C01365=2140.335600,108.803900,-378.952600,0.257831,3.013758,-90.000210
C01366=2142.949200,108.803900,-378.572900,0.601606,4.635229,-90.000210
C01367=2144.844900,108.803900,-378.971000,-2.778845,5.620716,-90.000210
C01368=2148.346300,108.803900,-378.603900,-0.275020,4.159674,-90.000210
C01369=2149.570000,108.803900,-378.482000,0.870896,2.818952,-90.000210
C01370=2153.470900,108.803900,-378.271600,-1.558445,6.233781,-90.000210
C01371=2155.140500,108.803900,-378.024400,-1.644389,3.477854,-90.000210
C01372=2158.623100,108.803900,-378.023900,-1.644389,8.823550,-90.000210
C01373=2159.706500,108.803900,-378.052300,0.200535,5.133702,-90.000210
C01374=2164.528500,108.803900,-377.988700,-3.924761,4.079460,-90.000210
C01375=2165.061600,108.803900,-377.750400,-1.799087,2.475178,-90.000210
C01376=2169.864400,108.803900,-377.381500,-2.503826,3.529420,-90.000210
C01377=2170.425300,108.803900,-377.373400,-0.068755,3.111161,-90.000210
C01378=2174.112300,108.803900,-377.090200,-0.693279,8.347995,-90.000210
C01379=2174.902100,108.803900,-377.071100,-2.457989,1.495420,-90.000210
C01380=2176.445800,108.803900,-376.837600,-1.151645,6.589015,-90.000210
C01381=2178.587100,108.803900,-377.080000,0.492744,5.546231,-90.000210
C01382=2179.426500,108.803900,-376.837800,-1.403747,4.159674,-90.000210
C01383=2180.476200,108.803900,-376.384800,-1.546986,8.342265,-90.000210
C01384=2181.164700,108.803900,-377.498800,-1.105809,12.839984,-90.000210
C01385=2185.019800,108.803900,-375.142900,-2.314749,16.489725,-90.000210
C01386=2185.530800,108.803900,-375.837200,-0.057296,11.768553,-90.000210
C01387=2188.541900,108.803900,-375.235400,-1.088620,-13.636396,-90.000210
C01388=2185.502100,58.803900,-375.622500,-0.051566,2.028271,-90.000210
C01389=2184.587500,58.803900,-375.704900,-1.157375,9.511099,-90.000210
C01390=2181.334500,58.803900,-375.888300,-0.120321,9.224621,-90.000210
C01391=2180.186000,58.803900,-376.104700,-1.346451,10.616908,-90.000210
C01392=2177.745200,58.803900,-376.686800,1.919409,5.872817,-90.000210
C01393=2175.909400,58.803900,-376.663100,-2.085566,0.280749,-90.000210
C01394=2174.454800,58.803900,-377.270400,-1.896490,10.530964,-90.000210
C01395=2172.787400,58.803900,-376.982500,0.509932,2.314749,-90.000210
C01396=2170.187600,58.803900,-377.417200,3.088243,5.930113,-90.000210
C01397=2168.929400,58.803900,-377.238000,0.807870,1.781899,-90.000210
C01398=2165.565800,58.803900,-377.616500,1.581364,7.792226,-90.000210
C01399=2164.422600,58.803900,-377.925700,0.401070,2.056918,-90.000210
C01400=2160.181900,58.803900,-377.880400,-3.472124,0.567228,-90.000210
C01401=2159.040000,58.803900,-378.155600,1.810547,3.787251,-90.000210
C01402=2155.756900,58.803900,-378.165400,0.618794,5.993139,-90.000210
C01403=2154.515100,58.803900,-378.187200,1.117268,-3.225752,-90.000210
C01404=2150.984900,58.803900,-378.776800,-0.452637,7.333860,-90.000210
C01405=2149.951300,58.803900,-378.829700,2.561121,2.457989,-90.000210
C01406=2145.683000,58.803900,-379.110300,1.793358,0.469825,-90.000210
C01407=2143.964500,58.803900,-379.252700,0.257831,2.045459,-90.000210
C01408=2140.681700,58.803900,-379.571700,-0.401070,3.638282,-90.000210
C01409=2139.364900,58.803900,-379.434900,-2.257454,2.566851,-90.000210
C01410=2135.250600,58.803900,-379.701700,0.166158,5.981679,-90.000210
C01411=2134.565900,58.803900,-379.901400,2.343397,2.274642,-90.000210
C01412=2130.555100,58.803900,-379.773400,0.974028,1.094349,-90.000210
C01413=2128.778000,58.803900,-380.055000,-1.346451,5.099324,-90.000210
C01414=2125.039800,58.803900,-379.997700,-2.005352,1.443854,-90.000210
C01415=2123.450000,58.803900,-380.182100,-2.354857,4.967544,-90.000210
C01416=2120.144500,58.803900,-380.051500,1.065701,4.967544,-90.000210
C01417=2119.439800,58.803900,-380.544400,-3.002299,6.841116,-90.000210
C01418=2115.315400,58.803900,-380.917300,-1.466772,2.755927,-90.000210
C01419=2114.666500,58.803900,-380.805000,-1.220400,4.417505,-90.000210
C01420=2110.782700,58.803900,-381.136300,0.051566,-0.148969,-90.000210
C01421=2109.540100,58.803900,-380.902600,1.226130,4.732631,-90.000210
C01422=2105.405600,58.803900,-381.373500,-0.974028,-0.515662,-90.000210
C01423=2104.154700,58.803900,-381.173700,-0.080214,3.386181,-90.000210
C01424=2100.313800,58.803900,-381.393300,1.443854,-2.939273,-90.000210
C01425=2099.416200,58.803900,-381.361500,3.197104,2.188699,-90.000210
C01426=2095.705700,58.803900,-381.541500,-0.865166,2.297561,-90.000210
C01427=2094.399000,58.803900,-381.243800,-1.902220,10.244485,-90.000210
C01428=2090.482500,58.803900,-381.699500,0.521392,0.538580,-90.000210
C01429=2089.894800,58.803900,-381.726800,-0.343775,7.093218,-90.000210
C01430=2088.622100,58.803900,-381.671700,-4.807116,3.311696,-90.000210
C01431=2085.713800,58.803900,-381.989400,2.509555,1.581364,-90.000210
C01432=2084.932900,58.803900,-382.119500,2.440800,-3.529420,-90.000210
C01433=2083.804500,58.803900,-382.023400,-3.036676,7.293753,-90.000210
C01434=2080.895000,58.803900,-382.327300,-6.864034,7.603150,-90.000210
C01435=2079.430100,58.803900,-382.144100,1.541256,0.137510,-90.000210
C01436=2076.700300,58.803900,-381.799600,-1.140186,-1.695955,-90.000210
C01437=2075.381200,58.803900,-381.594200,2.074107,2.641335,-90.000210
C01438=2074.734300,58.803900,-381.984200,-0.406800,10.204378,-90.000210
C01439=2073.666000,58.803900,-381.686800,1.077161,-1.747521,-90.000210
C01440=2070.998900,58.803900,-382.174100,-2.331938,5.580609,-90.000210
C01441=2069.894200,58.803900,-382.356100,0.022918,2.412152,-90.000210
C01442=2066.142600,58.803900,-381.817600,2.841871,-7.838063,-90.000210
C01443=2065.130800,58.803900,-382.222900,-0.000000,4.973274,-90.000210
C01444=2064.109000,58.803900,-382.313600,0.131780,0.045837,-90.000210
C01445=2059.976500,58.803900,-382.791600,0.017189,2.463719,-90.000210
C01446=2059.344800,58.803900,-382.491600,-1.621471,4.004975,-90.000210
C01447=2055.137600,58.803900,-382.767900,0.246372,0.928192,-90.000210
C01448=2054.262100,58.803900,-382.732000,-1.398017,9.608502,-90.000210
C01449=2050.756100,58.803900,-382.822700,-1.220400,1.799087,-90.000210
C01450=2049.656400,58.803900,-382.466400,-2.268913,4.755550,-90.000210
C01451=2045.238400,58.803900,-383.017300,0.349504,2.372045,-90.000210
C01452=2044.711100,58.803900,-382.562100,3.334614,0.177617,-90.000210
C01453=2040.460400,58.803900,-382.439700,-3.603905,-0.005730,-90.000210
C01454=2039.362700,58.803900,-382.724300,-3.804440,5.242564,-90.000210
C01455=2035.985300,58.803900,-382.893100,0.527121,2.538203,-90.000210
C01456=2034.820500,58.803900,-382.546000,1.346451,3.810169,-90.000210
C01457=2030.644000,58.803900,-382.672600,0.859437,-1.008406,-90.000210
C01458=2030.169900,58.803900,-383.193200,1.621471,1.134456,-90.000210
C01459=2025.187800,58.803900,-382.877900,-0.097403,-1.787628,-90.000210
C01460=2024.574700,58.803900,-383.229400,-0.074485,4.004975,-90.000210
C01461=2020.476400,58.803900,-383.039200,-7.431263,2.692902,-90.000210
C01462=2019.466600,58.803900,-382.959500,2.807493,-3.930490,-90.000210
C01463=2015.631800,58.803900,-382.903800,-2.286102,1.432394,-90.000210
C01464=2015.048100,58.803900,-382.657200,-0.315127,-0.956840,-90.000210
C01465=2010.573400,58.803900,-383.196100,0.435448,-0.481285,-90.000210
C01466=2010.196000,58.803900,-383.078200,1.575634,2.429341,-90.000210
C01467=2005.701400,58.803900,-383.121800,-0.022918,-0.418259,-90.000210
C01468=2004.681200,58.803900,-382.914000,1.650118,-0.464096,-90.000210
C01469=2000.403900,58.803900,-383.270500,2.016811,0.676090,-90.000210
C01470=1999.773000,58.803900,-382.763200,1.363640,-2.314749,-90.000210
C01471=1995.965500,58.803900,-383.525800,1.793358,1.266237,-90.000210
C01472=1994.614700,58.803900,-383.090400,-2.326209,3.873195,-90.000210
C01473=1990.010100,58.803900,-383.727900,2.349127,1.186023,-90.000210
C01474=1989.339500,58.803900,-382.844700,-7.906818,2.383504,-90.000210
C01475=1985.330500,58.803900,-383.000600,-1.541256,4.222699,-90.000210
C01476=1984.855800,58.803900,-383.668700,0.275020,-0.085944,-90.000210
C01477=1980.565200,58.803900,-383.301100,1.713144,0.309397,-90.000210
C01478=1979.406900,58.803900,-383.427700,-3.621093,-0.916732,-90.000210
C01479=1975.633400,58.803900,-383.409200,0.733386,3.426288,-90.000210
C01480=1974.632600,58.803900,-383.625600,-3.472124,-1.008406,-90.000210
C01481=1970.094700,58.803900,-383.404200,-0.297938,3.351803,-90.000210
C01482=1969.228600,58.803900,-383.285200,0.807870,-1.804817,-90.000210
C01483=1965.431900,58.803900,-383.353900,0.985487,0.681820,-90.000210
C01484=1964.322300,58.803900,-383.483100,0.418259,-0.859437,-90.000210
C01485=1960.406200,58.803900,-383.682400,-0.343775,5.815522,-90.000210
C01486=1959.568000,58.803900,-383.464300,0.544310,1.638659,-90.000210
C01487=1955.232300,58.803900,-383.720300,-1.707414,0.166158,-90.000210
C01488=1954.550100,58.803900,-384.072200,0.229183,0.166158,-90.000210
C01489=1950.253700,58.803900,-383.661000,-2.142862,3.959138,-90.000210
C01490=1949.237000,58.803900,-383.741700,-0.991217,-0.796411,-90.000210
C01491=1945.042300,58.803900,-383.696800,0.893814,2.830412,-90.000210
C01492=1944.229400,58.803900,-383.864500,-0.103132,-1.512609,-90.000210
C01493=1940.243800,58.803900,-383.674600,0.853707,0.223454,-90.000210
C01494=1939.598200,58.803900,-383.521800,-2.899166,0.721927,-90.000210
C01495=1934.733400,58.803900,-383.900000,1.180293,0.710468,-90.000210
C01496=1934.150000,58.803900,-383.736200,2.543933,-1.220400,-90.000210
C01497=1929.731700,58.803900,-383.984300,1.650118,-1.088620,-90.000210
C01498=1928.887000,58.803900,-383.919500,1.615741,2.320479,-90.000210
C01499=1925.319200,58.803900,-384.022700,1.294885,0.974028,-90.000210
C01500=1924.421800,58.803900,-383.615600,-0.269290,0.320856,-90.000210
C01501=1920.347700,58.803900,-383.889100,-2.509555,-2.217347,-90.000210
C01502=1918.947700,58.803900,-383.934000,-1.329262,2.979381,-90.000210
C01503=1915.472500,58.803900,-383.526300,2.985110,-2.629876,-90.000210
C01504=1914.276600,58.803900,-383.502500,1.844924,4.486260,-90.000210
C01505=1910.641200,58.803900,-383.604500,-0.395341,-1.466772,-90.000210
C01506=1908.610300,58.803900,-383.777400,0.790682,2.916355,-90.000210
C01507=1904.933000,58.803900,-383.473900,2.326209,0.378152,-90.000210
C01508=1903.988800,58.803900,-383.867400,1.260507,-4.383127,-90.000210
C01509=1899.603400,58.803900,-383.901900,0.211994,-1.203211,-90.000210
C01510=1899.065900,58.803900,-383.767000,-3.466395,-0.664631,-90.000210
C01511=1894.408000,58.803900,-383.572600,-0.996947,0.154699,-90.000210
C01512=1893.986600,58.803900,-383.686900,1.312073,-1.426665,-90.000210
C01513=1890.113800,58.803900,-383.601400,-2.532473,-3.655471,-90.000210
C01514=1885.581400,58.803900,-383.341900,-0.595876,-1.294885,-90.000210
C01515=1885.101800,58.803900,-383.330600,-3.283048,0.360963,-90.000210
C01516=1881.620200,58.803900,-382.819500,1.867842,-2.074107,-90.000210
C01517=1879.575800,58.803900,-383.315200,-2.738738,-4.887330,-90.000210
C01518=1875.961700,58.803900,-383.349800,0.240642,0.063025,-90.000210
C01519=1875.053400,58.803900,-383.258900,-1.105809,1.438124,-90.000210
C01520=1871.217400,58.803900,-383.091600,0.487014,0.847978,-90.000210
C01521=1870.023400,58.803900,-382.821900,-4.852953,-4.520637,-90.000210
C01522=1865.779800,58.803900,-382.711700,-2.028271,-3.305966,-90.000210
C01523=1864.214900,58.803900,-382.880300,0.326586,-1.770440,-90.000210
C01524=1860.166900,58.803900,-382.494200,-1.930868,-0.303668,-90.000210
C01525=1859.143500,58.803900,-382.129700,1.655848,-4.600851,-90.000210
C01526=1856.059600,58.803900,-382.618300,-0.790682,-1.191752,-90.000210
C01527=1854.337100,58.803900,-381.870600,2.005352,1.054242,-90.000210
C01528=1852.620800,58.803900,-382.149500,-0.131780,-5.414451,-90.000210
C01529=1850.548500,58.803900,-382.288500,-0.372423,-3.111161,-90.000210
C01530=1849.250100,58.803900,-382.128200,3.552338,-3.792981,-90.000210
C01531=1847.930100,58.803900,-381.849900,2.263183,-4.480530,-90.000210
C01532=1845.672200,58.803900,-381.812800,-2.223076,-3.838817,-90.000210
C01533=1844.518400,58.803900,-381.759500,-1.054242,-5.786874,-90.000210
C01534=1842.170400,58.803900,-381.737900,0.137510,-1.730333,-90.000210
C01535=1839.610700,58.803900,-381.495500,-0.383882,-3.036676,-90.000210
C01536=1835.873400,58.803900,-381.287400,-0.200535,-4.148214,-90.000210
C01537=1834.250800,58.803900,-381.223900,-0.143239,-4.795657,-90.000210
C01538=1830.424200,58.803900,-381.145200,1.541256,-4.715443,-90.000210
C01539=1829.330400,58.803900,-380.908500,-0.120321,-3.242941,-90.000210
C01540=1825.463600,58.803900,-380.787400,2.727279,-5.345696,-90.000210
C01541=1824.811300,58.803900,-380.790700,0.446907,-3.781521,-90.000210
C01542=1820.697200,58.803900,-380.122400,-4.411775,-2.309020,-90.000210
C01543=1820.073100,58.803900,-380.341800,-1.346451,-3.787251,-90.000210
C01544=1815.208000,58.803900,-379.935100,1.128727,-0.721927,-90.000210
C01545=1813.968500,58.803900,-379.830700,-3.122620,-1.781899,-90.000210
C01546=1810.175300,58.803900,-379.725400,-3.432017,-5.042029,-90.000210
C01547=1809.588700,58.803900,-379.670400,0.847978,-6.038975,-90.000210
C01548=1805.581100,58.803900,-379.087200,-0.458366,-7.156243,-90.000210
C01549=1804.197100,58.803900,-379.105600,4.469071,-6.978626,-90.000210
C01550=1800.624100,58.803900,-378.792900,1.546986,-3.552338,-90.000210
C01551=1800.080000,58.803900,-378.764800,-2.091296,-5.798333,-90.000210
C01552=1795.146200,58.803900,-377.697500,1.472502,-12.330052,-90.000210
C01553=1798.894300,8.803900,-378.601800,-3.489313,-5.557691,-90.000210
C01554=1799.874700,8.803900,-378.703700,-0.905273,-2.790304,-90.000210
C01555=1803.731800,8.803900,-378.851500,-0.527121,-8.542801,-90.000210
C01556=1804.996400,8.803900,-379.130200,1.117268,-9.419426,-90.000210
C01557=1808.212300,8.803900,-379.516200,0.452637,-4.996192,-90.000210
C01558=1810.246100,8.803900,-379.250100,1.002676,-4.365938,-90.000210
C01559=1813.388800,8.803900,-379.809400,-6.302536,0.773493,-90.000210
C01560=1814.666500,8.803900,-379.843100,1.403747,-3.506502,-90.000210
C01561=1817.731100,8.803900,-379.844200,1.518338,-4.308643,-90.000210
C01562=1819.765400,8.803900,-380.143400,1.369369,-0.435448,-90.000210
C01563=1823.736000,8.803900,-380.365700,0.647442,-3.426288,-90.000210
C01564=1825.030000,8.803900,-380.140400,-0.200535,-2.801764,-90.000210
C01565=1829.030600,8.803900,-381.056800,1.294885,-3.724226,-90.000210
C01566=1830.159200,8.803900,-380.847200,0.956840,-3.397640,-90.000210
C01567=1833.665900,8.803900,-381.235100,-1.386558,2.492366,-90.000210
C01568=1834.861100,8.803900,-381.245300,2.841871,-0.750575,-90.000210
C01569=1838.641500,8.803900,-381.487400,1.667307,-4.537826,-90.000210
C01570=1839.725400,8.803900,-381.101400,-1.655848,-0.458366,-90.000210
C01571=1840.896800,8.803900,-381.998000,-2.704361,-9.499640,-90.000210
C01572=1844.249100,8.803900,-381.278200,-1.707414,-1.644389,-90.000210
C01573=1845.828700,8.803900,-381.090700,-0.446907,-2.956462,-90.000210
C01574=1848.645500,8.803900,-381.508500,1.684496,-4.772738,-90.000210
C01575=1849.939500,8.803900,-381.733100,1.758980,2.097026,-90.000210
C01576=1851.853300,8.803900,-381.959200,-0.068755,-1.352180,-90.000210
C01577=1854.092400,8.803900,-382.227200,-0.223454,-2.097026,-90.000210
C01578=1855.033800,8.803900,-381.980700,-1.254778,-1.203211,-90.000210
C01579=1858.951100,8.803900,-381.746000,4.726902,-0.561499,-90.000210
C01580=1860.353300,8.803900,-382.463600,-0.303668,-3.093972,-90.000210
C01581=1861.721700,8.803900,-382.169600,2.022541,0.045837,-90.000210
C01582=1865.128600,8.803900,-382.819200,3.466395,-3.575257,-90.000210
C01583=1866.119700,8.803900,-381.824800,-0.000000,2.435071,-90.000210
C01584=1869.238400,8.803900,-383.038200,0.309397,-4.159674,-90.000210
C01585=1869.781300,8.803900,-382.206600,3.208564,-1.438124,-90.000210
C01586=1874.067800,8.803900,-382.729800,2.137133,2.973651,-90.000210
C01587=1874.982700,8.803900,-382.825800,0.068755,-0.544310,-90.000210
C01588=1877.430700,8.803900,-382.695100,1.415206,-1.976704,-90.000210
C01589=1880.280300,8.803900,-382.513300,-0.876625,-1.690225,-90.000210
C01590=1881.633900,8.803900,-382.741000,-2.629876,-3.575257,-90.000210
C01591=1884.822300,8.803900,-383.129700,-0.338045,-0.962569,-90.000210
C01592=1886.160000,8.803900,-382.472300,-1.546986,2.142862,-90.000210
C01593=1890.121700,8.803900,-383.547500,1.524068,-0.647442,-90.000210
C01594=1891.232400,8.803900,-383.371900,1.002676,-2.320479,-90.000210
C01595=1895.136100,8.803900,-383.093500,-2.074107,0.790682,-90.000210
C01596=1896.427800,8.803900,-383.638300,3.970598,-3.477854,-90.000210
C01597=1899.180000,8.803900,-383.160600,0.068755,-1.254778,-90.000210
C01598=1900.888600,8.803900,-382.681400,3.134079,-2.870519,-90.000210
C01599=1904.903400,8.803900,-383.065000,1.249048,0.475555,-90.000210
C01600=1905.816200,8.803900,-382.772800,2.956462,-0.011459,-90.000210
C01601=1909.631700,8.803900,-382.819700,-2.647065,2.612688,-90.000210
C01602=1914.174000,8.803900,-382.556800,5.878547,0.372423,-90.000210
C01603=1915.668900,8.803900,-383.397100,4.348750,-1.575634,-90.000210
C01604=1918.191500,8.803900,-382.853800,-0.956840,0.412530,-90.000210
C01605=1920.545000,8.803900,-383.109600,1.581364,0.189076,-90.000210
C01606=1923.828600,8.803900,-383.561000,-0.326586,2.011082,-90.000210
C01607=1925.621600,8.803900,-383.491300,2.818952,0.693279,-90.000210
C01608=1928.924300,8.803900,-383.132100,4.153944,2.480907,-90.000210
C01609=1930.221500,8.803900,-383.050700,3.586716,-0.676090,-90.000210
C01610=1934.139500,8.803900,-382.735300,1.976704,0.991217,-90.000210
C01611=1935.506700,8.803900,-382.861000,4.451882,-4.927437,-90.000210
C01612=1938.911000,8.803900,-382.668700,5.712389,3.242941,-90.000210
C01613=1939.988300,8.803900,-382.986500,2.079837,-6.858305,-90.000210
C01614=1944.067300,8.803900,-382.539000,0.515662,-1.019865,-90.000210
C01615=1945.073200,8.803900,-381.750700,3.472124,-2.394964,-90.000210
C01616=1948.562000,8.803900,-383.489800,5.826981,-3.884654,-90.000210
C01617=1949.549500,8.803900,-383.018800,-0.739116,1.799087,-90.000210
C01618=1951.671600,8.803900,-381.909100,2.876248,0.607335,-90.000210
C01619=1954.708200,8.803900,-382.811500,-0.464096,1.008406,-90.000210
C01620=1956.281200,8.803900,-382.140300,1.506879,-0.017189,-90.000210
C01621=1959.804800,8.803900,-382.649900,-0.143239,3.552338,-90.000210
C01622=1960.634200,8.803900,-382.671200,3.919031,3.019488,-90.000210
C01623=1964.757100,8.803900,-383.227900,1.552716,0.859437,-90.000210
C01624=1965.783600,8.803900,-382.461700,-0.206265,1.564175,-90.000210
C01625=1969.332500,8.803900,-382.489900,-2.515285,-1.753251,-90.000210
C01626=1970.399000,8.803900,-382.187200,4.486260,1.495420,-90.000210
C01627=1974.685600,8.803900,-382.745700,2.154321,3.036676,-90.000210
C01628=1975.213800,8.803900,-382.463300,2.755927,-0.051566,-90.000210
C01629=1979.096500,8.803900,-383.224900,-0.572958,6.216592,-90.000210
C01630=1980.965400,8.803900,-382.278900,5.219646,-0.813600,-90.000210
C01631=1983.944900,8.803900,-382.980900,-3.460665,2.904896,-90.000210
C01632=1985.069100,8.803900,-383.157900,2.194428,-5.305589,-90.000210
C01633=1988.765800,8.803900,-382.456300,-0.234913,-2.028271,-90.000210
C01634=1989.888800,8.803900,-382.090400,1.856383,1.432394,-90.000210
C01635=1990.341500,8.803900,-382.930800,1.409476,4.996192,-90.000210
C01636=1993.928900,8.803900,-382.864700,-0.756304,-2.830412,-90.000210
C01637=1995.346700,8.803900,-383.412200,2.807493,4.268536,-90.000210
C01638=1999.376500,8.803900,-382.764300,4.635229,4.555014,-90.000210
C01639=1999.957200,8.803900,-382.491700,1.478231,1.352180,-90.000210
C01640=2001.129100,8.803900,-381.640100,-6.130648,0.487014,-90.000210
C01641=2003.744400,8.803900,-383.015300,-6.291077,4.056541,-90.000210
C01642=2005.057700,8.803900,-382.069000,-0.687549,6.881223,-90.000210
C01643=2008.712000,8.803900,-382.085600,4.812845,1.403747,-90.000210
C01644=2009.806200,8.803900,-382.878700,-0.481285,5.076406,-90.000210
C01645=2012.925600,8.803900,-381.918700,-1.856383,-0.968299,-90.000210
C01646=2015.064200,8.803900,-382.624000,1.438124,-0.189076,-90.000210
C01647=2016.149900,8.803900,-382.482500,-4.320102,4.440423,-90.000210
C01648=2018.113800,8.803900,-382.473600,4.566474,2.973651,-90.000210
C01649=2019.538000,8.803900,-382.127700,1.340721,2.309020,-90.000210
C01650=2020.615000,8.803900,-382.598900,-0.103132,-2.853330,-90.000210
C01651=2023.397600,8.803900,-381.921300,2.268913,6.864034,-90.000210
C01652=2025.430500,8.803900,-381.853800,-0.452637,8.823550,-90.000210
C01653=2026.143200,8.803900,-382.299400,-1.094349,-6.170755,-90.000210
C01654=2029.744600,8.803900,-381.628100,3.506502,-0.080214,-90.000210
C01655=2030.943400,8.803900,-382.368600,1.329262,-2.320479,-90.000210
C01656=2033.843600,8.803900,-381.831700,-4.915978,1.059972,-90.000210
C01657=2035.120700,8.803900,-381.854300,3.191375,1.632930,-90.000210
C01658=2036.216200,8.803900,-381.666200,2.664254,1.254778,-90.000210
C01659=2039.656600,8.803900,-382.222300,2.114214,1.037054,-90.000210
C01660=2040.336700,8.803900,-382.027300,4.623769,3.930490,-90.000210
C01661=2044.682000,8.803900,-381.296300,0.974028,0.750575,-90.000210
C01662=2045.132200,8.803900,-382.311400,1.157375,2.549662,-90.000210
C01663=2046.168000,8.803900,-382.433100,-0.922462,0.716197,-90.000210
C01664=2049.178300,8.803900,-382.426800,0.905273,7.431263,-90.000210
C01665=2050.186200,8.803900,-381.789600,1.650118,3.878924,-90.000210
C01666=2051.798900,8.803900,-381.716500,0.481285,5.958761,-90.000210
C01667=2053.688400,8.803900,-382.030900,1.724603,2.137133,-90.000210
C01668=2054.878700,8.803900,-381.594000,1.363640,2.784575,-90.000210
C01669=2056.375300,8.803900,-381.770500,0.951110,0.137510,-90.000210
C01670=2058.327500,8.803900,-381.651900,2.675713,-5.867088,-90.000210
C01671=2059.785600,8.803900,-382.200000,0.154699,-0.269290,-90.000210
C01672=2061.250400,8.803900,-381.756800,3.214293,2.114214,-90.000210
C01673=2063.874300,8.803900,-382.207100,-3.644012,1.569904,-90.000210
C01674=2065.184100,8.803900,-382.199200,0.721927,-0.825059,-90.000210
C01675=2066.546900,8.803900,-382.027600,1.564175,-0.080214,-90.000210
C01676=2069.277800,8.803900,-381.350500,-1.226130,-1.449583,-90.000210
C01677=2070.702300,8.803900,-381.843300,0.979758,4.102378,-90.000210
C01678=2071.873400,8.803900,-381.587100,-0.028648,7.522936,-90.000210
C01679=2074.360300,8.803900,-381.986800,1.334992,2.561121,-90.000210
C01680=2075.422300,8.803900,-381.676700,2.011082,7.786496,-90.000210
C01681=2078.932700,8.803900,-381.534300,3.145538,-1.002676,-90.000210
C01682=2079.949400,8.803900,-381.507400,2.635606,-5.305589,-90.000210
C01683=2084.420700,8.803900,-381.675300,4.354479,-3.844547,-90.000210
C01684=2085.146700,8.803900,-381.581600,1.913679,2.985110,-90.000210
C01685=2087.746400,8.803900,-381.366900,0.498473,-0.229183,-90.000210
C01686=2089.249100,8.803900,-380.882100,1.770440,2.859059,-90.000210
C01687=2090.194300,8.803900,-382.156400,2.773116,2.372045,-90.000210
C01688=2094.465100,8.803900,-380.936300,-2.423611,2.945003,-90.000210
C01689=2096.081700,8.803900,-381.151500,2.257454,-1.380828,-90.000210
C01690=2099.895500,8.803900,-381.059100,1.042783,-0.951110,-90.000210
C01691=2101.198000,8.803900,-380.864700,2.372045,9.516829,-90.000210
C01692=2105.068100,8.803900,-381.276200,4.062271,4.360209,-90.000210
C01693=2106.438600,8.803900,-380.837900,-0.613065,1.655848,-90.000210
C01694=2109.528900,8.803900,-380.861000,0.704738,1.449583,-90.000210
C01695=2110.846600,8.803900,-380.588700,0.108862,7.041651,-90.000210
C01696=2114.640100,8.803900,-380.177100,-0.217724,2.503826,-90.000210
C01697=2115.458000,8.803900,-380.384400,-0.017189,6.205133,-90.000210
C01698=2119.588600,8.803900,-379.801400,1.088620,1.220400,-90.000210
C01699=2121.498600,8.803900,-379.873500,2.847600,2.354857,-90.000210
C01700=2124.614600,8.803900,-379.701300,-0.297938,0.103132,-90.000210
C01701=2126.311200,8.803900,-379.634300,1.363640,6.686417,-90.000210
C01702=2130.106600,8.803900,-379.760800,0.802141,2.309020,-90.000210
C01703=2133.256100,8.803900,-379.607200,-1.140186,3.082513,-90.000210
C01704=2135.454200,8.803900,-379.716100,1.466772,5.603527,-90.000210
C01705=2138.900600,8.803900,-379.399900,-0.974028,1.856383,-90.000210
C01706=2140.496400,8.803900,-379.454700,1.827735,1.902220,-90.000210
C01707=2143.219500,8.803900,-379.253800,-1.134456,5.614986,-90.000210
C01708=2144.888700,8.803900,-378.834900,-3.197104,6.652040,-90.000210
C01709=2148.266900,8.803900,-379.009800,2.274642,2.102755,-90.000210
C01710=2149.837900,8.803900,-378.563700,0.704738,0.779223,-90.000210
C01711=2154.077000,8.803900,-378.213200,1.558445,4.589392,-90.000210
C01712=2155.082100,8.803900,-378.577300,-0.063025,6.543178,-90.000210
C01713=2158.906100,8.803900,-377.860000,-1.873572,3.374721,-90.000210
C01714=2160.225200,8.803900,-378.014100,-1.948057,3.093972,-90.000210
C01715=2163.890600,8.803900,-377.623900,0.647442,5.614986,-90.000210
C01716=2164.880600,8.803900,-377.783800,1.621471,3.844547,-90.000210
C01717=2169.386500,8.803900,-377.358800,-4.262806,2.074107,-90.000210
C01718=2170.175100,8.803900,-377.246600,-1.489690,0.383882,-90.000210
C01719=2171.774900,8.803900,-376.772400,-2.796034,6.193674,-90.000210
C01720=2174.349300,8.803900,-377.086400,0.017189,4.658147,-90.000210
C01721=2175.360200,8.803900,-377.013800,1.913679,6.674958,-90.000210
C01722=2177.008300,8.803900,-377.163000,-7.454181,1.896490,-90.000210
C01723=2180.561900,8.803900,-376.316900,-0.171887,10.043950,-90.000210
C01724=2181.078100,8.803900,-376.110500,-2.286102,5.076406,-90.000210
C01725=2184.526000,8.803900,-375.725500,-4.314372,8.307888,-90.000210
C01726=2185.880000,-41.196100,-375.195400,-1.117268,8.600097,-90.000210
C01727=2184.495800,-41.196100,-375.702000,-1.524068,7.448451,-90.000210
C01728=2181.254800,-41.196100,-376.002700,-1.180293,5.133702,-90.000210
C01729=2179.901600,-41.196100,-376.252500,-4.881600,5.953031,-90.000210
C01730=2177.291700,-41.196100,-376.736900,-0.504203,5.431640,-90.000210
C01731=2174.987800,-41.196100,-377.102500,-0.263561,6.405668,-90.000210
C01732=2173.467500,-41.196100,-377.244300,-0.017189,6.365561,-90.000210
C01733=2170.873200,-41.196100,-376.921900,-0.349504,3.712767,-90.000210
C01734=2169.363500,-41.196100,-377.460900,-0.211994,7.127595,-90.000210
C01735=2166.065700,-41.196100,-377.214200,1.438124,5.500395,-90.000210
C01736=2165.275200,-41.196100,-377.323000,0.108862,3.432017,-90.000210
C01737=2163.485000,-41.196100,-377.080300,0.819330,6.331184,-90.000210
C01738=2160.102500,-41.196100,-377.738500,1.197482,2.916355,-90.000210
C01739=2158.853300,-41.196100,-377.593900,-1.128727,2.068378,-90.000210
C01740=2155.073000,-41.196100,-378.064900,1.369369,1.925138,-90.000210
C01741=2153.724200,-41.196100,-377.850000,1.352180,2.028271,-90.000210
C01742=2150.349000,-41.196100,-378.400400,0.762034,2.979381,-90.000210
C01743=2149.136700,-41.196100,-377.910500,3.116890,3.678389,-90.000210
C01744=2145.160300,-41.196100,-378.700300,1.655848,3.168457,-90.000210
C01745=2144.326800,-41.196100,-378.466200,1.690225,3.919031,-90.000210
C01746=2140.135800,-41.196100,-378.318400,-1.025594,1.145916,-90.000210
C01747=2138.981500,-41.196100,-379.103600,0.011459,2.068378,-90.000210
C01748=2135.291100,-41.196100,-378.850600,3.271589,3.071054,-90.000210
C01749=2133.841500,-41.196100,-379.406100,0.171887,0.177617,-90.000210
C01750=2130.488700,-41.196100,-378.890300,4.148214,2.584040,-90.000210
C01751=2128.923200,-41.196100,-379.018600,1.799087,7.356778,-90.000210
C01752=2125.737900,-41.196100,-379.393600,3.489313,0.452637,-90.000210
C01753=2123.975700,-41.196100,-378.591300,2.595499,1.839195,-90.000210
C01754=2120.075600,-41.196100,-379.170500,-0.607335,2.309020,-90.000210
C01755=2118.901600,-41.196100,-379.712800,0.916732,4.818575,-90.000210
C01756=2114.735000,-41.196100,-380.002700,-3.317426,-0.126051,-90.000210
C01757=2113.577900,-41.196100,-379.959100,2.962192,-3.260130,-90.000210
C01758=2110.098400,-41.196100,-379.433600,10.227297,3.867465,-90.000210
C01759=2109.561500,-41.196100,-379.487300,3.197104,-2.429341,-90.000210
C01760=2105.376800,-41.196100,-380.509000,4.744091,3.500772,-90.000210
C01761=2104.898100,-41.196100,-379.374400,1.443854,2.967921,-90.000210
C01762=2100.737400,-41.196100,-379.764200,1.352180,-0.045837,-90.000210
C01763=2099.790300,-41.196100,-380.834500,-1.472502,0.229183,-90.000210
C01764=2095.224100,-41.196100,-380.131200,4.612310,2.750197,-90.000210
C01765=2093.930100,-41.196100,-380.331700,1.604282,7.585961,-90.000210
C01766=2089.893200,-41.196100,-380.417300,3.397640,4.761279,-90.000210
C01767=2089.258900,-41.196100,-380.773800,0.779223,-1.925138,-90.000210
C01768=2085.330100,-41.196100,-380.757400,0.790682,0.819330,-90.000210
C01769=2083.879100,-41.196100,-379.511000,3.019488,-1.398017,-90.000210
C01770=2079.836600,-41.196100,-380.416000,0.624524,0.315127,-90.000210
C01771=2079.038700,-41.196100,-380.368400,2.056918,-1.879302,-90.000210
C01772=2074.672000,-41.196100,-379.861700,3.798710,2.498096,-90.000210
C01773=2074.092400,-41.196100,-380.658000,7.047381,8.244863,-90.000210
C01774=2070.056600,-41.196100,-379.715000,-0.464096,3.156997,-90.000210
C01775=2069.076500,-41.196100,-380.400900,-0.326586,-1.277696,-90.000210
C01776=2065.277900,-41.196100,-380.250600,-0.567228,3.277319,-90.000210
C01777=2063.880600,-41.196100,-379.731600,2.251724,-1.380828,-90.000210
C01778=2060.201500,-41.196100,-379.972500,1.163104,-1.231859,-90.000210
C01779=2059.099600,-41.196100,-380.740700,8.227674,1.380828,-90.000210
C01780=2055.123100,-41.196100,-380.849500,3.288778,0.349504,-90.000210
C01781=2053.996000,-41.196100,-380.050500,6.755172,-2.223076,-90.000210
C01782=2049.819700,-41.196100,-380.443700,5.935843,-0.068755,-90.000210
C01783=2049.134800,-41.196100,-381.700300,0.022918,5.660823,-90.000210
C01784=2045.224000,-41.196100,-381.245000,5.523313,1.959516,-90.000210
C01785=2044.771200,-41.196100,-380.905500,-4.027893,-0.074485,-90.000210
C01786=2040.257500,-41.196100,-381.458500,1.094349,4.463341,-90.000210
C01787=2039.336100,-41.196100,-379.745600,0.888085,1.753251,-90.000210
C01788=2035.560200,-41.196100,-380.149800,0.727656,-3.237212,-90.000210
C01789=2033.515600,-41.196100,-381.337000,1.014135,-2.773116,-90.000210
C01790=2029.970400,-41.196100,-381.111700,4.875871,2.091296,-90.000210
C01791=2028.017600,-41.196100,-380.702300,0.750575,-0.905273,-90.000210
C01792=2025.281000,-41.196100,-380.401200,5.380074,-0.429718,-90.000210
C01793=2023.851300,-41.196100,-380.213200,0.481285,-2.435071,-90.000210
C01794=2019.728100,-41.196100,-380.300400,2.412152,-2.400693,-90.000210
C01795=2019.058600,-41.196100,-381.536000,1.764710,2.595499,-90.000210
C01796=2014.946900,-41.196100,-380.978700,1.186023,-0.487014,-90.000210
C01797=2010.390000,-41.196100,-380.567500,-1.638659,5.334237,-90.000210
C01798=2009.731700,-41.196100,-381.456000,3.964868,1.506879,-90.000210
C01799=2006.217700,-41.196100,-381.020200,0.154699,3.993516,-90.000210
C01800=2004.385900,-41.196100,-380.094900,1.220400,2.790304,-90.000210
C01801=2001.248400,-41.196100,-381.863700,6.669229,5.082136,-90.000210
C01802=2000.379500,-41.196100,-380.943500,5.586339,0.550039,-90.000210
C01803=1997.761400,-41.196100,-382.132400,2.211617,-0.171887,-90.000210
C01804=1995.113800,-41.196100,-381.971700,0.257831,3.105431,-90.000210
C01805=1994.652900,-41.196100,-379.974000,2.188699,1.707414,-90.000210
C01806=1989.787700,-41.196100,-381.076400,2.217347,-1.122997,-90.000210
C01807=1989.016100,-41.196100,-379.930100,2.349127,0.389611,-90.000210
C01808=1986.291800,-41.196100,-381.148200,-1.168834,-0.704738,-90.000210
C01809=1984.627600,-41.196100,-380.667900,5.746767,2.343397,-90.000210
C01810=1980.711100,-41.196100,-381.395000,3.093972,-0.481285,-90.000210
C01811=1980.047300,-41.196100,-381.569600,2.016811,-4.279995,-90.000210
C01812=1976.640500,-41.196100,-382.374000,6.972896,-1.340721,-90.000210
C01813=1975.100000,-41.196100,-380.121300,-2.784575,0.137510,-90.000210
C01814=1973.698600,-41.196100,-381.294000,-0.080214,5.609257,-90.000210
C01815=1970.010500,-41.196100,-380.203500,9.316294,-2.515285,-90.000210
C01816=1968.613500,-41.196100,-382.095800,-1.031324,1.844924,-90.000210
C01817=1966.022300,-41.196100,-381.592700,3.999245,2.543933,-90.000210
C01818=1964.655500,-41.196100,-380.029600,2.131403,1.839195,-90.000210
C01819=1960.547600,-41.196100,-380.255200,2.165780,1.718873,-90.000210
C01820=1959.422400,-41.196100,-380.031900,8.519882,-1.867842,-90.000210
C01821=1957.473800,-41.196100,-382.205800,3.099702,-0.779223,-90.000210
C01822=1955.043700,-41.196100,-381.735600,4.394586,0.137510,-90.000210
C01823=1954.062100,-41.196100,-381.684000,6.554637,1.541256,-90.000210
C01824=1950.141700,-41.196100,-380.586400,4.795657,0.825059,-90.000210
C01825=1949.476100,-41.196100,-381.977900,1.816276,-8.233404,-90.000210
C01826=1945.507800,-41.196100,-381.667900,1.277696,5.792603,-90.000210
C01827=1944.984400,-41.196100,-381.700800,3.386181,2.412152,-90.000210
C01828=1943.695100,-41.196100,-382.237100,-0.011459,2.377775,-90.000210
C01829=1941.079500,-41.196100,-381.081000,1.804817,4.463341,-90.000210
C01830=1939.451900,-41.196100,-380.357700,0.538580,3.781521,-90.000210
C01831=1935.406000,-41.196100,-381.487800,2.228806,-1.690225,-90.000210
C01832=1934.176300,-41.196100,-380.632300,5.746767,-0.762034,-90.000210
C01833=1930.488600,-41.196100,-381.185900,6.159296,-2.417882,-90.000210
C01834=1929.880500,-41.196100,-381.659800,-1.684496,0.492744,-90.000210
C01835=1926.074600,-41.196100,-380.394200,0.842248,4.211240,-90.000210
C01836=1924.491200,-41.196100,-380.870900,6.972896,-0.097403,-90.000210
C01837=1920.888500,-41.196100,-380.599800,4.320102,4.148214,-90.000210
C01838=1920.372900,-41.196100,-381.287800,7.058840,-6.858305,-90.000210
C01839=1919.171800,-41.196100,-382.295300,0.005730,2.446530,-90.000210
C01840=1915.534400,-41.196100,-381.857100,-6.995815,13.229595,-90.000210
C01841=1914.581800,-41.196100,-381.964100,10.513776,-7.540125,-90.000210
C01842=1910.831800,-41.196100,-382.252200,3.884654,-4.182592,-90.000210
C01843=1909.397200,-41.196100,-381.109400,5.804062,0.441178,-90.000210
C01844=1905.433200,-41.196100,-381.982500,5.265482,-2.922085,-90.000210
C01845=1904.354100,-41.196100,-380.850500,4.153944,-1.157375,-90.000210
C01846=1901.224700,-41.196100,-380.146500,1.191752,2.784575,-90.000210
C01847=1900.943200,-41.196100,-382.312100,1.340721,-1.581364,-90.000210
C01848=1898.677700,-41.196100,-381.742100,-0.922462,1.323533,-90.000210
C01849=1895.878500,-41.196100,-381.910800,3.609634,-0.063025,-90.000210
C01850=1895.638900,-41.196100,-380.243000,2.039730,1.541256,-90.000210
C01851=1892.807100,-41.196100,-382.261800,0.962569,0.200535,-90.000210
C01852=1890.565400,-41.196100,-380.594800,1.707414,1.157375,-90.000210
C01853=1889.860500,-41.196100,-381.233100,-0.796411,-1.059972,-90.000210
C01854=1885.286500,-41.196100,-382.385700,0.578687,1.426665,-90.000210
C01855=1884.612900,-41.196100,-380.791100,1.294885,-0.945380,-90.000210
C01856=1882.779800,-41.196100,-382.009500,3.684119,1.037054,-90.000210
C01857=1880.149700,-41.196100,-381.749400,2.372045,-5.930113,-90.000210
C01858=1878.438900,-41.196100,-380.761600,0.951110,-0.360963,-90.000210
C01859=1875.006800,-41.196100,-382.215600,1.306344,-5.093595,-90.000210
C01860=1874.154300,-41.196100,-381.613200,-1.059972,-0.859437,-90.000210
C01861=1870.916000,-41.196100,-381.373000,1.770440,3.489313,-90.000210
C01862=1869.849000,-41.196100,-381.316300,-0.653172,0.389611,-90.000210
C01863=1866.246500,-41.196100,-382.056300,-1.684496,-6.222322,-90.000210
C01864=1864.858600,-41.196100,-379.990200,2.824682,1.776169,-90.000210
C01865=1864.164300,-41.196100,-381.007400,3.002299,0.767763,-90.000210
C01866=1859.806200,-41.196100,-380.511900,1.610011,0.767763,-90.000210
C01867=1859.069300,-41.196100,-381.389300,0.252101,-0.292208,-90.000210
C01868=1854.817700,-41.196100,-379.850200,0.148969,4.612310,-90.000210
C01869=1853.868500,-41.196100,-381.034700,5.890006,-1.432394,-90.000210
C01870=1850.003000,-41.196100,-380.905800,2.647065,-0.515662,-90.000210
C01871=1848.676900,-41.196100,-380.548000,0.773493,1.993893,-90.000210
C01872=1844.734500,-41.196100,-380.810200,-1.420935,0.595876,-90.000210
C01873=1844.143200,-41.196100,-380.694600,-1.650118,-0.985487,-90.000210
C01874=1840.047100,-41.196100,-379.707900,4.451882,-5.947302,-90.000210
C01875=1838.314100,-41.196100,-379.343200,1.363640,-3.025217,-90.000210
C01876=1834.393000,-41.196100,-379.620000,-2.108485,0.338045,-90.000210
C01877=1833.918600,-41.196100,-380.668100,2.274642,-6.193674,-90.000210
C01878=1829.774100,-41.196100,-379.832000,-0.744845,-2.452259,-90.000210
C01879=1825.669200,-41.196100,-379.624900,6.497341,-3.890383,-90.000210
C01880=1825.187900,-41.196100,-379.253200,3.082513,-5.236834,-90.000210
C01881=1820.708000,-41.196100,-378.938300,2.687172,-3.013758,-90.000210
C01882=1819.044900,-41.196100,-379.962500,-0.446907,1.312073,-90.000210
C01883=1815.594300,-41.196100,-379.344100,3.019488,-0.922462,-90.000210
C01884=1814.615800,-41.196100,-378.950900,3.432017,-2.813223,-90.000210
C01885=1810.688100,-41.196100,-379.312300,-0.166158,-2.102755,-90.000210
C01886=1809.855000,-41.196100,-379.145700,4.285724,-2.767386,-90.000210
C01887=1805.671400,-41.196100,-378.925600,0.292208,-3.374721,-90.000210
C01888=1804.704000,-41.196100,-378.996200,2.360586,-4.549285,-90.000210
C01889=1800.366600,-41.196100,-378.306200,4.320102,-5.832710,-90.000210
C01890=1799.418300,-41.196100,-378.526600,-5.294130,-12.639449,-90.000210
C01891=1795.305000,-91.196100,-377.541600,1.054242,7.110406,-90.000210
C01892=1799.418900,-91.196100,-377.424900,1.816276,-5.271212,-90.000210
C01893=1800.080400,-91.196100,-377.530100,-0.899544,-6.113460,-90.000210
C01894=1804.178900,-91.196100,-377.422000,0.527121,-1.163104,-90.000210
C01895=1805.558800,-91.196100,-378.041700,2.727279,-4.079460,-90.000210
C01896=1809.552100,-91.196100,-378.343400,-0.922462,3.099702,-90.000210
C01897=1810.802700,-91.196100,-377.922800,2.280372,-1.403747,-90.000210
C01898=1814.674800,-91.196100,-377.946100,-0.217724,2.154321,-90.000210
C01899=1816.221700,-91.196100,-377.447600,4.027893,1.140186,-90.000210
C01900=1819.459700,-91.196100,-378.316500,0.624524,-1.449583,-90.000210
C01901=1820.188300,-91.196100,-378.633200,3.919031,-3.775792,-90.000210
C01902=1823.981900,-91.196100,-378.201500,0.498473,0.578687,-90.000210
C01903=1825.225300,-91.196100,-377.414900,3.603905,0.572958,-90.000210
C01904=1829.473200,-91.196100,-377.953500,3.689848,0.211994,-90.000210
C01905=1830.985100,-91.196100,-378.696500,-0.790682,0.830789,-90.000210
C01906=1834.377800,-91.196100,-377.651000,1.850654,3.254400,-90.000210
C01907=1835.959000,-91.196100,-377.260400,0.464096,-0.956840,-90.000210
C01908=1839.694900,-91.196100,-377.295500,2.492366,-0.521392,-90.000210
C01909=1840.541800,-91.196100,-378.454700,2.950733,-6.239510,-90.000210
C01910=1844.696300,-91.196100,-377.160200,0.194806,2.406423,-90.000210
C01911=1845.955400,-91.196100,-377.972800,3.580986,-0.074485,-90.000210
C01912=1848.927700,-91.196100,-378.948900,6.514530,-2.142862,-90.000210
C01913=1849.965600,-91.196100,-377.457300,4.451882,1.151645,-90.000210
C01914=1851.787800,-91.196100,-376.910400,4.325831,-2.394964,-90.000210
C01915=1854.842300,-91.196100,-377.542100,1.140186,2.750197,-90.000210
C01916=1855.268200,-91.196100,-378.573400,2.669983,-0.378152,-90.000210
C01917=1859.702800,-91.196100,-378.097700,3.048135,0.378152,-90.000210
C01918=1860.339600,-91.196100,-377.126900,1.483961,4.893060,-90.000210
C01919=1864.837400,-91.196100,-377.522500,2.160051,-1.587093,-90.000210
C01920=1866.502900,-91.196100,-378.692900,-1.993893,1.432394,-90.000210
C01921=1869.655800,-91.196100,-379.088500,5.271212,0.280749,-90.000210
C01922=1870.902400,-91.196100,-378.347700,3.792981,3.747144,-90.000210
C01923=1874.608700,-91.196100,-378.370400,7.127595,-2.721550,-90.000210
C01924=1875.701800,-91.196100,-377.271200,2.469448,1.896490,-90.000210
C01925=1879.089700,-91.196100,-376.878100,2.452259,0.189076,-90.000210
C01926=1880.404400,-91.196100,-377.206400,2.291831,-0.022918,-90.000210
C01927=1883.226300,-91.196100,-379.326300,1.976704,-3.036676,-90.000210
C01928=1884.972800,-91.196100,-378.617500,0.395341,1.409476,-90.000210
C01929=1889.337000,-91.196100,-377.344200,5.259753,-0.739116,-90.000210
C01930=1890.538400,-91.196100,-377.879400,3.672659,0.888085,-90.000210
C01931=1894.036400,-91.196100,-376.879800,1.294885,2.360586,-90.000210
C01932=1895.783700,-91.196100,-378.730600,7.998491,-2.549662,-90.000210
C01933=1899.291000,-91.196100,-379.024600,3.517961,0.515662,-90.000210
C01934=1900.259300,-91.196100,-378.071800,3.002299,-0.280749,-90.000210
C01935=1902.386500,-91.196100,-377.434900,4.234158,-4.274265,-90.000210
C01936=1905.020700,-91.196100,-378.297300,11.659691,4.205510,-90.000210
C01937=1907.374900,-91.196100,-379.871200,1.965245,2.245995,-90.000210
C01938=1909.572800,-91.196100,-377.869600,1.483961,1.896490,-90.000210
C01939=1910.710100,-91.196100,-377.032900,4.050812,-1.758980,-90.000210
C01940=1914.960000,-91.196100,-379.427400,4.784198,0.578687,-90.000210
C01941=1915.743200,-91.196100,-378.526000,1.323533,-1.529797,-90.000210
C01942=1920.119800,-91.196100,-379.065500,4.491989,1.529797,-90.000210
C01943=1920.959300,-91.196100,-378.296100,-0.022918,4.761279,-90.000210
C01944=1924.741400,-91.196100,-380.206700,2.240265,0.756304,-90.000210
C01945=1925.292200,-91.196100,-378.183400,2.675713,-5.105054,-90.000210
C01946=1930.023700,-91.196100,-377.070400,6.520260,3.271589,-90.000210
C01947=1930.189000,-91.196100,-378.390900,5.884277,1.128727,-90.000210
C01948=1934.079100,-91.196100,-376.687200,-2.383504,0.836518,-90.000210
C01949=1935.446400,-91.196100,-379.999500,3.506502,1.082890,-90.000210
C01950=1938.838100,-91.196100,-377.816600,2.635606,-0.968299,-90.000210
C01951=1940.436500,-91.196100,-378.391900,4.434693,1.615741,-90.000210
C01952=1942.886800,-91.196100,-379.959800,0.693279,2.211617,-90.000210
C01953=1944.917200,-91.196100,-377.943600,4.279995,1.936597,-90.000210
C01954=1948.261700,-91.196100,-377.396700,3.059595,1.546986,-90.000210
C01955=1949.956200,-91.196100,-378.329400,1.334992,0.498473,-90.000210
C01956=1953.464800,-91.196100,-377.372700,3.517961,-1.673037,-90.000210
C01957=1955.037100,-91.196100,-379.269300,1.936597,2.796034,-90.000210
C01958=1957.644200,-91.196100,-377.607800,1.747521,2.268913,-90.000210
C01959=1959.560500,-91.196100,-379.741500,2.578310,7.580232,-90.000210
C01960=1963.395800,-91.196100,-378.215300,7.746389,0.441178,-90.000210
C01961=1964.946600,-91.196100,-376.641700,3.764333,-0.853707,-90.000210
C01962=1969.099700,-91.196100,-378.729000,5.105054,1.850654,-90.000210
C01963=1970.306000,-91.196100,-377.055900,3.741414,-0.183346,-90.000210
C01964=1972.157200,-91.196100,-376.780300,0.779223,1.558445,-90.000210
C01965=1974.946500,-91.196100,-378.646700,2.715820,-0.269290,-90.000210
C01966=1975.717600,-91.196100,-379.977300,7.035922,0.876625,-90.000210
C01967=1979.866700,-91.196100,-378.788600,-0.475555,-0.825059,-90.000210
C01968=1981.044900,-91.196100,-377.480900,2.291831,0.464096,-90.000210
C01969=1984.927400,-91.196100,-379.068600,4.560744,0.658901,-90.000210
C01970=1987.335300,-91.196100,-376.378000,4.205510,2.349127,-90.000210
C01971=1990.373300,-91.196100,-378.245900,3.008028,1.426665,-90.000210
C01972=1992.305200,-91.196100,-379.490600,2.423611,0.796411,-90.000210
C01973=1994.371000,-91.196100,-379.740700,6.079082,0.550039,-90.000210
C01974=1995.503400,-91.196100,-379.443200,0.492744,-1.776169,-90.000210
C01975=1999.561100,-91.196100,-377.473300,1.518338,2.217347,-90.000210
C01976=2000.080400,-91.196100,-379.228000,1.289155,2.962192,-90.000210
C01977=2004.406500,-91.196100,-378.900800,-1.650118,2.068378,-90.000210
C01978=2005.652800,-91.196100,-377.941400,2.618417,0.802141,-90.000210
C01979=2009.434900,-91.196100,-378.794300,0.423989,-3.449206,-90.000210
C01980=2010.261000,-91.196100,-377.289600,2.836141,-0.624524,-90.000210
C01981=2013.853400,-91.196100,-379.442200,2.962192,4.211240,-90.000210
C01982=2015.071400,-91.196100,-377.219300,2.658524,2.240265,-90.000210
C01983=2019.320600,-91.196100,-379.177000,3.781521,-0.584417,-90.000210
C01984=2020.278600,-91.196100,-377.598200,4.491989,3.122620,-90.000210
C01985=2024.061700,-91.196100,-378.312600,1.936597,2.601228,-90.000210
C01986=2024.673200,-91.196100,-377.500200,5.746767,1.048513,-90.000210
C01987=2028.765600,-91.196100,-377.287400,3.838817,-5.471747,-90.000210
C01988=2029.403200,-91.196100,-379.302600,-2.234535,-1.306344,-90.000210
C01989=2033.995500,-91.196100,-379.271100,2.927814,1.724603,-90.000210
C01990=2035.196000,-91.196100,-377.121800,4.818575,0.452637,-90.000210
C01991=2036.257100,-91.196100,-376.721200,10.152812,2.372045,-90.000210
C01992=2040.109900,-91.196100,-378.754900,7.935465,0.550039,-90.000210
C01993=2041.225700,-91.196100,-377.911800,-0.441178,1.065701,-90.000210
C01994=2044.180500,-91.196100,-379.373200,2.933544,-1.638659,-90.000210
C01995=2044.990600,-91.196100,-377.271000,1.352180,4.016434,-90.000210
C01996=2049.316800,-91.196100,-379.066800,6.302536,-1.266237,-90.000210
C01997=2050.431000,-91.196100,-379.407900,0.578687,1.386558,-90.000210
C01998=2054.812800,-91.196100,-378.624300,0.223454,0.962569,-90.000210
C01999=2055.478200,-91.196100,-377.232100,6.399939,-2.635606,-90.000210
C02000=2059.087800,-91.196100,-379.472500,4.182592,1.122997,-90.000210
C02001=2060.348900,-91.196100,-379.251500,4.486260,4.904519,-90.000210
C02002=2064.525700,-91.196100,-377.693900,3.432017,0.252101,-90.000210
C02003=2065.787700,-91.196100,-377.027100,1.930868,-1.472502,-90.000210
C02004=2067.675200,-91.196100,-377.871200,5.030569,-0.063025,-90.000210
C02005=2069.595700,-91.196100,-376.894300,2.469448,1.243318,-90.000210
C02006=2070.674500,-91.196100,-378.584300,6.594744,2.005352,-90.000210
C02007=2074.375000,-91.196100,-378.345800,4.039352,-0.802141,-90.000210
C02008=2075.996200,-91.196100,-378.574200,2.956462,-0.635983,-90.000210
C02009=2079.628700,-91.196100,-379.307200,-2.131403,-1.518338,-90.000210
C02010=2080.836600,-91.196100,-378.302200,5.683741,1.907949,-90.000210
C02011=2084.764200,-91.196100,-378.169000,-0.693279,0.114592,-90.000210
C02012=2086.437400,-91.196100,-376.636800,5.597798,-1.203211,-90.000210
C02013=2089.410600,-91.196100,-378.030400,0.876625,3.156997,-90.000210
C02014=2090.183700,-91.196100,-377.411000,2.864789,3.111161,-90.000210
C02015=2094.448800,-91.196100,-378.114000,2.303290,-0.590147,-90.000210
C02016=2096.058400,-91.196100,-377.332100,1.976704,2.859059,-90.000210
C02017=2099.543700,-91.196100,-377.890000,6.016057,0.338045,-90.000210
C02018=2100.315200,-91.196100,-378.222700,3.953409,-0.429718,-90.000210
C02019=2104.184400,-91.196100,-376.632700,5.202457,-2.377775,-90.000210
C02020=2104.790700,-91.196100,-377.159400,2.664254,0.080214,-90.000210
C02021=2107.833200,-91.196100,-376.917600,4.354479,1.667307,-90.000210
C02022=2110.286500,-91.196100,-378.242200,5.930113,1.059972,-90.000210
C02023=2111.691200,-91.196100,-377.226200,4.365938,6.210862,-90.000210
C02024=2114.634200,-91.196100,-378.486600,0.796411,-1.552716,-90.000210
C02025=2116.213000,-91.196100,-378.735700,6.715065,2.457989,-90.000210
C02026=2119.530700,-91.196100,-376.715100,0.945380,-0.057296,-90.000210
C02027=2121.044100,-91.196100,-377.621900,1.913679,2.309020,-90.000210
C02028=2124.313900,-91.196100,-377.459900,4.463341,4.245617,-90.000210
C02029=2125.062700,-91.196100,-377.243200,4.171133,-1.289155,-90.000210
C02030=2128.421800,-91.196100,-376.976900,5.242564,3.357533,-90.000210
C02031=2129.559200,-91.196100,-377.491600,1.827735,3.947679,-90.000210
C02032=2131.041700,-91.196100,-378.289500,2.297561,4.658147,-90.000210
C02033=2134.586000,-91.196100,-377.315700,2.773116,2.509555,-90.000210
C02034=2135.602800,-91.196100,-377.583700,1.816276,2.538203,-90.000210
C02035=2138.526500,-91.196100,-377.954700,1.008406,4.302913,-90.000210
C02036=2140.068800,-91.196100,-376.562000,2.303290,4.491989,-90.000210
C02037=2141.212700,-91.196100,-376.416200,1.203211,6.147837,-90.000210
C02038=2144.686800,-91.196100,-376.860700,0.744845,1.896490,-90.000210
C02039=2145.499300,-91.196100,-376.622900,1.134456,0.423989,-90.000210
C02040=2149.245900,-91.196100,-377.512500,3.151268,1.420935,-90.000210
C02041=2150.530400,-91.196100,-376.290900,2.687172,1.965245,-90.000210
C02042=2154.261200,-91.196100,-375.625400,1.781899,4.171133,-90.000210
C02043=2155.389400,-91.196100,-377.406900,-0.532851,5.500395,-90.000210
C02044=2158.923700,-91.196100,-376.796100,3.042406,2.102755,-90.000210
C02045=2159.995500,-91.196100,-377.108300,2.188699,5.380074,-90.000210
C02046=2162.658000,-91.196100,-377.093500,-2.927814,1.277696,-90.000210
C02047=2165.115800,-91.196100,-376.774200,-1.145916,1.976704,-90.000210
C02048=2166.465700,-91.196100,-376.259600,1.134456,0.320856,-90.000210
C02049=2169.854900,-91.196100,-376.573100,2.263183,3.609634,-90.000210
C02050=2171.046600,-91.196100,-376.056000,-0.452637,0.481285,-90.000210
C02051=2174.160400,-91.196100,-376.291000,4.027893,3.798710,-90.000210
C02052=2175.265900,-91.196100,-375.729000,4.239888,3.443476,-90.000210
C02053=2179.561800,-91.196100,-375.441200,-1.294885,4.681065,-90.000210
C02054=2180.555300,-91.196100,-376.351600,3.718496,6.697877,-90.000210
C02055=2184.038700,-91.196100,-375.049500,-0.945380,5.420181,-90.000210
C02056=2185.498200,-91.196100,-374.824100,6.537448,3.626823,-90.000210
C02057=2185.415100,-141.196100,-374.060000,2.669983,2.417882,-90.000210
C02058=2184.214300,-141.196100,-373.905800,3.838817,-0.532851,-90.000210
C02059=2180.012200,-141.196100,-374.573500,-0.275020,1.718873,-90.000210
C02060=2179.127200,-141.196100,-373.260600,4.841493,1.655848,-90.000210
C02061=2175.684200,-141.196100,-373.842900,2.807493,1.615741,-90.000210
C02062=2174.219500,-141.196100,-375.290800,0.120321,1.993893,-90.000210
C02063=2170.489300,-141.196100,-374.723500,0.750575,-0.143239,-90.000210
C02064=2169.134300,-141.196100,-375.269300,2.446530,0.882355,-90.000210
C02065=2165.315100,-141.196100,-373.747600,5.339967,2.945003,-90.000210
C02066=2164.630100,-141.196100,-375.232700,1.592823,-2.051189,-90.000210
C02067=2160.260500,-141.196100,-374.253400,3.248671,-0.475555,-90.000210
C02068=2159.387200,-141.196100,-375.240500,3.208564,2.320479,-90.000210
C02069=2155.362800,-141.196100,-374.889500,3.260130,2.337668,-90.000210
C02070=2154.922700,-141.196100,-375.396400,1.644389,-3.105431,-90.000210
C02071=2150.433100,-141.196100,-374.026600,6.611933,0.320856,-90.000210
C02072=2149.135500,-141.196100,-374.393900,2.435071,0.590147,-90.000210
C02073=2145.477900,-141.196100,-375.714300,3.735685,1.037054,-90.000210
C02074=2144.146800,-141.196100,-373.491100,9.551206,2.589769,-90.000210
C02075=2140.769500,-141.196100,-374.776700,5.024840,-0.292208,-90.000210
C02076=2139.289900,-141.196100,-373.542100,7.414074,-1.392287,-90.000210
C02077=2135.263800,-141.196100,-375.429800,7.351049,0.183346,-90.000210
C02078=2133.968100,-141.196100,-373.056800,1.088620,0.074485,-90.000210
C02079=2130.077900,-141.196100,-375.677200,3.540879,2.320479,-90.000210
C02080=2129.113500,-141.196100,-373.373200,6.107730,-0.360963,-90.000210
C02081=2125.272800,-141.196100,-375.578900,2.234535,-0.475555,-90.000210
C02082=2124.761100,-141.196100,-376.048200,2.383504,1.524068,-90.000210
C02083=2120.328000,-141.196100,-375.059200,4.279995,3.185645,-90.000210
C02084=2118.606900,-141.196100,-375.500900,2.904896,-1.340721,-90.000210
C02085=2115.318800,-141.196100,-372.750300,6.766632,5.305589,-90.000210
C02086=2113.745600,-141.196100,-375.727200,1.942327,2.211617,-90.000210
C02087=2110.355300,-141.196100,-376.311100,2.876248,2.664254,-90.000210
C02088=2109.416100,-141.196100,-375.774400,2.675713,1.214671,-90.000210
C02089=2105.001600,-141.196100,-375.638100,5.506124,-0.555769,-90.000210
C02090=2104.265800,-141.196100,-372.948600,9.539747,-1.541256,-90.000210
C02091=2100.516900,-141.196100,-375.890600,3.781521,0.320856,-90.000210
C02092=2099.725600,-141.196100,-375.017500,5.351426,2.595499,-90.000210
C02093=2095.436000,-141.196100,-374.505700,3.134079,-2.188699,-90.000210
C02094=2094.167300,-141.196100,-374.712900,7.396885,-1.472502,-90.000210
C02095=2090.205900,-141.196100,-375.986200,1.220400,-0.893814,-90.000210
C02096=2089.109700,-141.196100,-374.205600,4.131026,-2.171510,-90.000210
C02097=2085.580300,-141.196100,-375.997300,3.414828,-0.670361,-90.000210
C02098=2084.360700,-141.196100,-374.346000,4.772738,-0.349504,-90.000210
C02099=2080.253000,-141.196100,-373.722700,6.016057,1.690225,-90.000210
C02100=2079.835200,-141.196100,-376.286600,5.460288,1.100079,-90.000210
C02101=2074.913100,-141.196100,-376.787900,5.970220,-1.117268,-90.000210
C02102=2073.522100,-141.196100,-375.699100,5.305589,-0.292208,-90.000210
C02103=2069.173700,-141.196100,-373.234500,4.222699,0.928192,-90.000210
C02104=2066.401900,-141.196100,-374.355200,0.676090,1.936597,-90.000210
C02105=2064.927900,-141.196100,-375.525000,1.163104,1.449583,-90.000210
C02106=2061.460600,-141.196100,-375.886500,-0.991217,3.403369,-90.000210
C02107=2059.609800,-141.196100,-376.501600,3.964868,-1.449583,-90.000210
C02108=2055.666100,-141.196100,-376.502300,3.890383,0.338045,-90.000210
C02109=2055.045300,-141.196100,-375.888500,1.564175,-0.830789,-90.000210
C02110=2051.232500,-141.196100,-374.111300,-0.017189,1.529797,-90.000210
C02111=2049.797900,-141.196100,-376.208100,7.098947,1.128727,-90.000210
C02112=2046.719400,-141.196100,-376.168200,5.150891,1.713144,-90.000210
C02113=2045.239500,-141.196100,-372.335700,-0.492744,-0.360963,-90.000210
C02114=2041.406300,-141.196100,-374.903000,1.243318,1.203211,-90.000210
C02115=2039.762300,-141.196100,-374.660300,3.500772,0.229183,-90.000210
C02116=2036.008500,-141.196100,-373.939600,10.215837,2.801764,-90.000210
C02117=2034.926300,-141.196100,-373.407600,8.382373,-1.575634,-90.000210
C02118=2030.385500,-141.196100,-374.996300,4.595122,-1.019865,-90.000210
C02119=2029.826100,-141.196100,-374.272300,9.831956,-2.320479,-90.000210
C02120=2026.054900,-141.196100,-375.886700,3.535150,0.481285,-90.000210
C02121=2024.793500,-141.196100,-372.708000,0.933921,2.423611,-90.000210
C02122=2020.791600,-141.196100,-373.674200,11.699798,-2.945003,-90.000210
C02123=2019.172100,-141.196100,-375.199200,3.913302,-0.194806,-90.000210
C02124=2016.262900,-141.196100,-377.076700,2.784575,5.872817,-90.000210
C02125=2014.369600,-141.196100,-375.197200,2.372045,0.423989,-90.000210
C02126=2010.352800,-141.196100,-374.971500,4.681065,0.286479,-90.000210
C02127=2009.288200,-141.196100,-376.093000,6.050434,0.859437,-90.000210
C02128=2005.597400,-141.196100,-375.731900,5.678012,0.080214,-90.000210
C02129=2004.514200,-141.196100,-376.381900,6.589015,-0.578687,-90.000210
C02130=2000.011400,-141.196100,-373.316600,8.771984,4.503448,-90.000210
C02131=1998.643000,-141.196100,-376.369700,3.563797,-1.122997,-90.000210
C02132=1995.495000,-141.196100,-375.756200,6.147837,4.096648,-90.000210
C02133=1994.531200,-141.196100,-374.155600,9.425156,-1.501149,-90.000210
C02134=1990.070600,-141.196100,-375.098200,3.065324,-0.664631,-90.000210
C02135=1989.589500,-141.196100,-374.441000,5.660823,3.111161,-90.000210
C02136=1984.910300,-141.196100,-374.777500,0.807870,4.371668,-90.000210
C02137=1983.861200,-141.196100,-374.952900,4.297183,3.139809,-90.000210
C02138=1980.391400,-141.196100,-374.252200,6.056164,0.074485,-90.000210
C02139=1979.309700,-141.196100,-375.340600,3.861736,1.564175,-90.000210
C02140=1975.109500,-141.196100,-376.260300,6.205133,1.621471,-90.000210
C02141=1974.206500,-141.196100,-375.762200,3.053865,0.630254,-90.000210
C02142=1970.228800,-141.196100,-374.936100,2.142862,1.059972,-90.000210
C02143=1969.207600,-141.196100,-375.892800,6.869764,0.326586,-90.000210
C02144=1965.515000,-141.196100,-375.103000,3.592445,-0.968299,-90.000210
C02145=1964.102200,-141.196100,-376.394300,5.569150,-2.480907,-90.000210
C02146=1959.717200,-141.196100,-375.815700,4.251347,-0.853707,-90.000210
C02147=1959.054000,-141.196100,-373.895700,3.718496,3.076783,-90.000210
C02148=1954.785100,-141.196100,-374.983600,3.523690,0.085944,-90.000210
C02149=1954.384600,-141.196100,-375.969700,-0.423989,3.363262,-97.167912
C02150=1950.054900,-141.196100,-375.487600,2.429341,0.045837,-90.000210
C02151=1949.440100,-141.196100,-375.245900,4.056541,-0.911003,-90.000210
C02152=1945.526000,-141.196100,-376.724700,4.360209,-2.452259,-90.000210
C02153=1944.222500,-141.196100,-374.130000,9.602773,-4.010705,-90.000210
C02154=1940.229900,-141.196100,-376.375200,5.884277,1.690225,-90.000210
C02155=1939.527200,-141.196100,-377.085900,-0.108862,1.128727,-90.000210
C02156=1935.213100,-141.196100,-373.944100,3.586716,-1.965245,-90.000210
C02157=1934.819000,-141.196100,-375.337500,5.013381,1.105809,-90.000210
C02158=1930.636700,-141.196100,-375.890200,2.601228,0.040107,-90.000210
C02159=1929.735100,-141.196100,-376.410200,1.736062,0.200535,-90.000210
C02160=1925.900100,-141.196100,-375.823100,4.898789,-0.664631,-90.000210
C02161=1924.700500,-141.196100,-373.832900,4.669606,-0.681820,-90.000210
C02162=1920.470500,-141.196100,-376.522700,1.896490,1.483961,-90.000210
C02163=1919.832800,-141.196100,-376.398400,7.058840,-1.163104,-90.000210
C02164=1916.892300,-141.196100,-375.801400,5.030569,0.080214,-90.000210
C02165=1915.052000,-141.196100,-373.246600,1.375099,1.942327,-90.000210
C02166=1912.060800,-141.196100,-376.956500,4.979003,-0.630254,-90.000210
C02167=1910.298900,-141.196100,-375.968800,2.051189,1.541256,-90.000210
C02168=1908.582600,-141.196100,-376.159300,2.297561,3.919031,-90.000210
C02169=1905.388000,-141.196100,-373.909300,6.909871,-4.033623,-90.000210
C02170=1903.985300,-141.196100,-376.680200,3.231482,-0.825059,-90.000210
C02171=1900.049900,-141.196100,-376.768800,-0.309397,0.406800,-90.000210
C02172=1899.194200,-141.196100,-376.566600,4.738361,2.881978,-90.000210
C02173=1895.499600,-141.196100,-374.703300,3.271589,2.595499,-90.000210
C02174=1894.268200,-141.196100,-376.976300,1.524068,-1.535527,-90.000210
C02175=1890.500400,-141.196100,-375.186300,9.591313,3.008028,-90.000210
C02176=1889.495600,-141.196100,-376.046400,3.008028,0.103132,-90.000210
C02177=1885.342500,-141.196100,-376.640900,3.397640,-0.349504,-90.000210
C02178=1885.135300,-141.196100,-375.791200,3.151268,-0.916732,-90.000210
C02179=1879.748800,-141.196100,-375.833000,6.250970,-0.888085,-90.000210
C02180=1878.976300,-141.196100,-375.179100,7.608880,-2.423611,-90.000210
C02181=1875.506800,-141.196100,-376.619000,9.711635,-2.733009,-90.000210
C02182=1874.493600,-141.196100,-374.949800,6.050434,0.360963,-90.000210
C02183=1870.194200,-141.196100,-374.646200,5.254023,3.861736,-90.000210
C02184=1869.293000,-141.196100,-375.463700,3.036676,-0.498473,-90.000210
C02185=1865.075900,-141.196100,-376.316300,2.406423,1.678766,-90.000210
C02186=1864.404600,-141.196100,-375.624900,0.412530,2.337668,-90.000210
C02187=1859.803800,-141.196100,-375.872200,2.171510,0.492744,-90.000210
C02188=1858.398300,-141.196100,-375.605800,3.134079,-0.143239,-90.000210
C02189=1854.864000,-141.196100,-375.996800,3.076783,-0.085944,-90.000210
C02190=1853.834400,-141.196100,-374.837900,2.291831,1.426665,-90.000210
C02191=1850.410700,-141.196100,-375.284300,2.274642,3.008028,-90.000210
C02192=1849.748000,-141.196100,-375.547500,2.750197,1.117268,-90.000210
C02193=1845.055200,-141.196100,-375.674600,3.409099,5.712389,-90.000210
C02194=1844.434200,-141.196100,-377.106000,-3.764333,7.540125,-90.000210
C02195=1840.894700,-141.196100,-375.702800,1.306344,-0.733386,-90.000210
C02196=1839.805300,-141.196100,-376.567800,1.862113,1.581364,-90.000210
C02197=1835.935000,-141.196100,-377.111400,1.019865,-2.990840,-90.000210
C02198=1834.687700,-141.196100,-375.834300,8.296429,1.254778,-90.000210
C02199=1832.895400,-141.196100,-376.758400,1.902220,-0.521392,-90.000210
C02200=1829.331300,-141.196100,-375.944500,13.241055,2.830412,-90.000210
C02201=1825.616400,-141.196100,-376.772300,2.549662,-2.297561,-90.000210
C02202=1824.719900,-141.196100,-376.707800,-0.716197,2.423611,-90.000210
C02203=1823.375000,-141.196100,-376.275600,1.461042,2.595499,-90.000210
C02204=1820.148400,-141.196100,-376.699000,0.922462,1.902220,-90.000210
C02205=1819.386300,-141.196100,-377.239300,-0.733386,7.941195,-90.000210
C02206=1817.633800,-141.196100,-377.017400,-4.079460,7.620339,-90.000210
C02207=1815.194000,-141.196100,-377.208900,0.922462,0.320856,-90.000210
C02208=1813.793700,-141.196100,-377.163800,2.074107,-0.527121,-90.000210
C02209=1810.514800,-141.196100,-376.879400,1.037054,0.458366,-90.000210
C02210=1809.304000,-141.196100,-376.514000,5.603527,5.935843,-90.000210
C02211=1805.917100,-141.196100,-377.286100,1.443854,1.701685,-90.000210
C02212=1805.150600,-141.196100,-377.071100,-1.312073,3.139809,-90.000210
C02213=1803.613600,-141.196100,-376.936400,4.835764,-1.019865,-90.000210
C02214=1800.646400,-141.196100,-376.815200,1.741792,1.747521,-90.000210
C02215=1799.896800,-141.196100,-377.079600,-1.002676,0.120321,-90.000210
C02216=1798.042100,-141.196100,-377.026000,0.108862,5.448829,-90.000210
C02217=1794.253600,-141.196100,-377.324400,1.718873,11.252891,-90.000210
C02218=1812.109500,341.105500,-503.612600,89.811134,-0.234913,0.000000
C02219=2127.650500,341.132200,-503.612600,90.578898,-0.275020,-0.000000
C02220=2159.023800,341.159900,-503.612600,90.607546,-0.492744,-0.005730
C02221=1816.234900,341.190300,-503.612600,89.604870,0.154699,-0.000000
C02222=1821.738400,341.222100,-503.612600,90.000210,0.068755,-0.000000
C02223=1812.786700,341.237100,-503.612600,89.455901,-0.292208,0.000000
C02224=1809.568300,341.249200,-503.612600,83.164824,0.521392,-0.063025
C02225=1831.712400,341.267300,-503.612600,89.662165,0.492744,-0.005730
C02226=1826.384500,341.287600,-503.612600,89.547574,0.211994,-0.000000
C02227=1835.441800,341.299400,-503.612600,89.730920,0.114592,-0.000000
C02228=1840.177200,341.323100,-503.612600,89.673625,0.458366,-0.000000
C02229=1835.884800,341.334600,-503.612600,89.879889,0.240642,-0.000000
C02230=2119.313000,341.341300,-503.612600,89.633517,0.148969,-0.000000
C02231=2152.042800,341.346000,-503.612600,90.830999,0.022918,0.000000
C02232=2175.237500,341.354800,-503.612600,90.040318,0.406800,0.000000
C02233=1808.484300,341.385900,-503.612600,89.616329,-1.002676,0.005730
C02234=2144.675900,341.398100,-503.612600,90.859647,-0.280749,-0.005730
C02235=1798.586600,341.407200,-503.612600,89.639247,0.836518,-0.005730
C02236=1838.296800,341.417000,-503.612600,89.536115,-0.767763,0.005730
C02237=2112.907800,341.440300,-503.612600,90.951320,-0.784952,-0.011459
C02238=2136.688000,341.448700,-503.612600,90.962780,-0.275020,-0.005730
C02239=2090.048400,341.463900,-503.612600,91.025805,-0.166158,-0.005730
C02240=1866.740500,341.476100,-503.612600,84.093016,-0.034377,0.005730
C02241=2119.757400,341.491000,-503.612600,90.756515,-0.355234,-0.005730
C02242=1858.245800,341.509100,-503.612600,90.452847,0.458366,0.005730
C02243=2166.766400,341.523700,-503.612600,90.939861,0.538580,0.011459
C02244=1851.449100,341.538300,-503.612600,90.670571,0.842248,0.011459
C02245=2144.147600,341.553500,-503.612600,90.601816,-0.229183,-0.000000
C02246=1829.104800,341.580700,-503.612600,86.476520,0.532851,-0.034377
C02247=1861.433200,341.584600,-503.612600,89.639247,0.446907,-0.000000
C02248=2184.909600,341.594700,-503.612600,89.581951,1.913679,-0.011459
C02249=2091.279500,341.606500,-503.612600,90.991427,-1.002676,-0.017189
C02250=1817.924600,341.619000,-503.612600,88.751162,4.308643,-0.091673
C02251=2128.544600,341.634900,-503.612600,75.258006,0.401070,-0.103132
C02252=2189.650900,341.644700,-503.612600,91.678977,-4.606581,-0.137510
C02253=2117.508600,341.652500,-503.612600,90.412740,-0.309397,-0.000000
C02254=2109.284300,341.657500,-503.612600,89.650706,-0.721927,0.005730
C02255=2090.436700,341.673400,-503.612600,91.879512,0.034377,0.000000
C02256=2114.097000,341.679800,-503.612600,90.269501,-0.211994,-0.000000
C02257=2126.105100,341.684600,-503.612600,91.191963,0.412530,0.011459
C02258=2089.212200,341.696000,-503.612600,89.799675,-0.561499,0.000000
C02259=1866.067800,341.706200,-503.612600,89.897078,0.870896,-0.000000
C02260=2127.724100,341.717700,-503.612600,90.767974,0.137510,0.000000
C02261=2081.920700,341.730500,-503.612600,90.733596,-1.145916,-0.017189
C02262=2079.389300,341.738100,-503.612600,90.028858,-0.452637,-0.000000
C02263=1876.495600,341.751100,-503.612600,89.421523,1.025594,-0.011459
C02264=1875.989500,341.764000,-503.612600,77.355032,0.446907,-0.103132
C02265=2183.623100,341.792300,-503.612600,90.584627,1.701685,0.017189
C02266=2072.497100,341.803500,-503.612600,90.206475,-0.401070,-0.000000
C02267=2080.170300,341.818000,-503.612600,90.412740,-0.418259,-0.005730
C02268=1887.562600,341.829500,-503.612600,90.080425,1.002676,0.000000
C02269=2189.014800,341.847700,-503.612600,89.793946,-3.873195,0.011459
C02270=2076.462800,341.853500,-503.612600,89.593410,-0.676090,0.005730
C02271=2063.601500,341.860600,-503.612600,89.925726,-0.584417,0.000000
C02272=1880.479800,341.880200,-503.612600,90.011670,1.174563,0.000000
C02273=2072.651300,341.889500,-503.612600,90.326796,-0.183346,-0.000000
C02274=2142.630000,341.920400,-503.612600,91.438335,0.641713,0.017189
C02275=2163.746800,341.939300,-503.612600,82.620514,0.888085,-0.114592
C02276=2043.757000,341.950400,-503.612600,90.028858,0.211994,0.000000
C02277=2143.560600,341.978800,-503.612600,80.592243,0.418259,-0.068755
C02278=2152.254400,341.994400,-503.612600,86.407765,-0.991217,0.063025
C02279=1890.422400,342.008600,-503.612600,89.232447,0.888085,-0.011459
C02280=2187.978400,342.021900,-503.612600,93.644222,-0.240642,-0.017189
C02281=1997.694900,342.034600,-503.612600,88.837106,-8.176108,0.166158
C02282=1909.060200,342.052800,-503.612600,90.853918,1.082890,0.017189
C02283=1902.578300,342.072400,-503.612600,89.742379,0.641713,-0.005730
C02284=1894.728000,342.089300,-503.612600,90.137720,1.375099,0.005730
C02285=2088.376600,342.092800,-503.612600,86.367658,-2.045459,0.131780
C02286=1919.373700,342.116300,-503.612600,88.963157,1.271966,-0.022918
C02287=1998.261000,342.133700,-503.612600,87.536492,-1.982434,0.085944
C02288=1997.057700,342.151800,-503.612600,89.026182,-0.332316,0.005730
C02289=1985.819400,342.166700,-503.612600,83.359630,2.463719,-0.286479
C02290=1910.512600,342.177800,-503.612600,81.835562,0.229183,-0.034377
C02291=2049.023600,342.193400,-503.612600,90.533061,-0.045837,-0.000000
C02292=2036.066400,342.204500,-503.612600,90.235123,-0.555769,-0.000000
C02293=2032.569100,342.235600,-503.612600,89.748109,-0.240642,0.000000
C02294=1901.945000,342.245000,-503.612600,89.496008,1.048513,-0.011459
C02295=1912.115100,342.262700,-503.612600,89.129315,1.277696,-0.017189
C02296=2025.810400,342.269700,-503.612600,89.604870,0.074485,-0.000000
C02297=1898.412900,342.295000,-503.612600,86.476520,-0.847978,0.051566
C02298=2029.161400,342.309900,-503.612600,85.662920,-0.343775,0.028648
C02299=1902.070100,342.318400,-503.612600,90.120532,1.827735,0.005730
C02300=1927.560000,342.328800,-503.612600,88.928779,0.561499,-0.011459
C02301=2003.102000,342.352100,-503.612600,89.261095,-0.177617,0.000000
C02302=1982.107000,342.368000,-503.612600,90.212205,-0.567228,-0.000000
C02303=2008.875000,342.379200,-503.612600,89.306932,0.085944,-0.000000
C02304=2017.438000,342.392700,-503.612600,89.438712,-0.246372,0.000000
C02305=1928.227700,342.404500,-503.612600,83.835185,-0.085944,0.011459
C02306=1937.098800,342.419000,-503.612600,88.699596,-0.527121,0.011459
C02307=1942.371800,342.434900,-503.612600,88.413117,-0.005730,0.000000
C02308=1916.394300,342.451500,-503.612600,89.748109,0.555769,-0.000000
C02309=1942.013800,342.472400,-503.612600,89.450171,0.234913,-0.000000
C02310=1970.210400,342.503800,-503.612600,89.003264,-0.194806,0.005730
C02311=1958.875000,342.539600,-503.612600,89.622058,-0.475555,0.005730
C02312=1953.389600,342.556200,-503.612600,90.452847,-1.214671,-0.011459
C02313=1927.791100,342.573400,-503.612600,89.868430,0.383882,-0.000000
C02314=1936.371200,342.595700,-503.612600,90.080425,0.171887,0.000000
C02315=1927.557900,342.619600,-503.612600,89.937185,0.870896,-0.000000
C02316=1971.976400,342.660900,-503.612600,90.103343,-0.320856,-0.000000
C02317=1985.894000,342.701800,-503.612600,90.378363,0.080214,0.000000
C02318=1933.723800,342.718900,-503.612600,91.134667,0.807870,0.017189
C02319=1983.719200,342.754500,-503.612600,87.989129,-1.420935,0.051566
C02320=1967.433100,342.769700,-503.612600,88.917320,0.578687,-0.011459
C02321=1971.507500,342.796100,-503.612600,88.510520,0.126051,-0.005730
C02322=1978.383300,342.823400,-503.612600,89.564763,-0.057296,0.000000
C02323=1956.724200,342.919700,-503.612600,89.719461,-0.194806,0.000000
C02324=1964.207800,342.910600,-553.612600,89.455901,0.022918,-0.000000
C02325=1956.730900,342.867100,-553.612600,89.415794,0.733386,-0.005730
C02326=1949.078500,342.842700,-553.612600,90.332526,0.372423,0.000000
C02327=1964.487700,342.819700,-553.612600,90.097613,-1.059972,-0.000000
C02328=1980.017700,342.771400,-553.612600,90.298149,-0.733386,-0.005730
C02329=1979.608600,342.747100,-553.612600,90.808081,-0.091673,-0.000000
C02330=1991.957500,342.725100,-553.612600,90.000210,0.063025,0.000000
C02331=1961.526200,342.702200,-553.612600,89.897078,0.269290,-0.000000
C02332=1983.865300,342.684200,-553.612600,90.154909,-0.383882,-0.000000
C02333=1962.726300,342.669400,-553.612600,90.957050,-0.343775,-0.005730
C02334=1991.699800,342.655000,-553.612600,89.186610,-0.217724,0.005730
C02335=1935.378500,342.638300,-553.612600,90.750785,0.372423,0.005730
C02336=1989.062900,342.618000,-553.612600,89.937185,-0.011459,0.000000
C02337=1998.951400,342.595700,-553.612600,89.931456,-1.140186,0.000000
C02338=1957.989400,342.568700,-553.612600,90.916943,0.303668,0.005730
C02339=1958.395800,342.561300,-553.612600,91.421146,-0.022918,-0.000000
C02340=1912.496500,342.529900,-553.612600,90.470036,0.509932,0.005730
C02341=1994.182600,342.510700,-553.612600,91.913889,-0.194806,-0.005730
C02342=1980.976200,342.483900,-553.612600,91.203422,-0.309397,-0.005730
C02343=2004.766100,342.464300,-553.612600,90.303878,-1.432394,-0.005730
C02344=2003.375600,342.426800,-553.612600,90.510143,-0.635983,-0.005730
C02345=1952.385700,342.402800,-553.612600,91.782109,0.750575,0.022918
C02346=1910.094700,342.379200,-553.612600,90.361174,1.793358,0.011459
C02347=2015.315300,342.351500,-553.612600,91.191963,-1.300614,-0.028648
C02348=1938.235600,342.325500,-553.612600,91.386768,-0.240642,-0.005730
C02349=2013.285800,342.308200,-553.612600,90.848188,-0.807870,-0.011459
C02350=2019.297200,342.292300,-553.612600,89.604870,-0.693279,0.005730
C02351=2008.569300,342.270600,-553.612600,91.335202,-0.635983,-0.017189
C02352=2018.916400,342.222400,-553.612600,90.802351,-0.762034,-0.011459
C02353=1979.372100,342.200100,-553.612600,91.083101,-0.865166,-0.017189
C02354=2016.598500,342.168700,-553.612600,90.699219,-1.455313,-0.017189
C02355=2006.372200,342.140100,-553.612600,91.959726,-0.853707,-0.028648
C02356=2030.472900,342.119400,-553.612600,89.157963,-0.928192,0.011459
C02357=1890.291700,342.068400,-553.612600,90.000210,0.796411,0.000000
C02358=1897.591000,342.045400,-553.612600,91.243529,1.592823,0.034377
C02359=2045.790400,342.020700,-553.612600,89.301202,-0.418259,0.005730
C02360=2045.991900,341.966700,-553.612600,91.083101,-0.469825,-0.011459
C02361=2038.443800,341.945900,-553.612600,90.120532,-0.418259,-0.000000
C02362=2042.479600,341.930500,-553.612600,91.805028,-0.074485,-0.000000
C02363=1898.504200,341.915600,-553.612600,89.942915,1.827735,-0.000000
C02364=2032.882800,341.883700,-553.612600,91.764920,-1.426665,-0.045837
C02365=2015.277700,341.840600,-553.612600,91.289365,-1.180293,-0.028648
C02366=1898.244900,341.801500,-553.612600,91.432605,1.002676,0.022918
C02367=1893.562800,341.768000,-553.612600,90.750785,1.002676,0.011459
C02368=1880.777100,341.723800,-553.612600,90.481495,1.168834,0.011459
C02369=2046.840600,341.707200,-553.612600,90.160639,-0.825059,-0.000000
C02370=2069.878100,341.676100,-553.612600,90.916943,-0.842248,-0.011459
C02371=2040.561600,341.657200,-553.612600,91.902430,-0.985487,-0.034377
C02372=2052.105000,341.625800,-553.612600,90.813811,-0.693279,-0.011459
C02373=1875.965100,341.578100,-553.612600,90.813811,0.452637,0.005730
C02374=2082.093400,341.573100,-553.612600,91.541467,-1.151645,-0.028648
C02375=1799.023700,341.543000,-553.612600,90.687760,1.415206,0.017189
C02376=1860.945600,341.526800,-553.612600,89.828323,0.951110,-0.000000
C02377=2089.483100,341.518000,-553.612600,90.693489,-0.790682,-0.011459
C02378=1867.784400,341.508200,-553.612600,90.641923,0.246372,0.000000
C02379=1803.221900,341.494400,-553.612600,90.074695,-0.802141,-0.000000
C02380=1796.053400,341.486400,-553.612600,90.189287,7.110406,0.022918
C02381=1851.170600,341.469400,-553.612600,89.885619,0.567228,-0.000000
C02382=2071.772100,341.439600,-553.612600,90.905484,-1.352180,-0.022918
C02383=2066.800800,341.418300,-553.612600,91.002887,-1.037054,-0.017189
C02384=2185.746500,341.402500,-553.612600,89.816864,0.223454,-0.000000
C02385=1808.857900,341.395000,-553.612600,89.301202,-0.555769,0.005730
C02386=1861.348900,341.384600,-553.612600,89.942915,0.951110,-0.000000
C02387=1794.346900,341.374800,-553.612600,92.635816,14.289567,0.653172
C02388=2058.599500,341.362400,-553.612600,90.429929,-0.721927,-0.005730
C02389=2172.169600,341.353500,-553.612600,90.825270,0.401070,0.005730
C02390=2052.220800,341.343700,-553.612600,90.573168,-0.802141,-0.005730
C02391=1831.522400,341.336900,-553.612600,89.885619,-0.034377,0.000000
C02392=1806.243800,341.327100,-553.612600,89.690813,-0.395341,0.000000
C02393=2094.196100,341.319000,-553.612600,90.361174,-0.928192,-0.005730
C02394=1830.253700,341.299800,-553.612600,89.874160,-0.028648,0.000000
C02395=2095.532400,341.289300,-553.612600,91.174774,-1.409476,-0.028648
C02396=1836.079000,341.278800,-553.612600,90.011670,0.022918,0.000000
C02397=2177.034900,341.269700,-553.612600,90.372633,1.764710,0.011459
C02398=2070.756100,341.248400,-553.612600,91.065912,-0.670361,-0.011459
C02399=2178.247200,341.240600,-553.612600,90.143450,0.658901,0.000000
C02400=1860.429800,341.235200,-553.612600,90.745056,4.325831,0.057296
C02401=2155.399000,341.221700,-553.612600,91.071642,-0.177617,-0.005730
C02402=1850.372500,341.199800,-553.612600,90.475765,0.441178,0.005730
C02403=1794.823700,341.170700,-553.612600,90.790892,14.318215,0.194806
C02404=1827.853300,341.157500,-553.612600,90.613275,-0.292208,-0.005730
C02405=2165.438800,341.146400,-553.612600,90.361174,0.269290,0.000000
C02406=2170.953500,341.132500,-553.612600,90.429929,0.085944,0.000000
C02407=2090.251600,341.116600,-553.612600,90.177827,-0.561499,-0.000000
C02408=2079.914400,341.095000,-553.612600,90.888295,-0.550039,-0.005730
C02409=2163.450000,341.067000,-553.612600,90.630464,0.750575,0.005730
C02410=2079.593800,341.045000,-553.612600,90.160639,0.618794,0.000000
C02411=2103.730600,341.030200,-553.612600,91.438335,-0.383882,-0.011459
C02412=2173.328500,341.004100,-553.612600,90.355444,1.174563,0.005730
C02413=2096.643600,340.968700,-553.612600,90.338256,-0.246372,-0.000000
C02414=2115.653300,340.926800,-553.612600,90.464306,-0.572958,-0.005730
C02415=2172.555400,340.907900,-553.612600,90.808081,1.466772,0.022918
C02416=2166.320100,340.877300,-553.612600,90.727867,0.527121,0.005730
C02417=2102.683700,340.848400,-553.612600,90.871106,-0.956840,-0.017189
C02418=2159.266400,340.812600,-553.612600,89.948644,0.338045,-0.000000
C02419=2124.739500,340.747400,-553.612600,90.865377,0.051566,0.000000
C02420=2147.251400,340.711900,-553.612600,90.481495,-0.131780,-0.000000
C02421=2124.127400,340.644000,-553.612600,90.401281,-0.263561,-0.000000
C02422=2155.011400,340.515300,-553.612600,90.710678,0.922462,0.011459
C02423=2135.657000,340.072400,-603.612600,90.699219,0.739116,0.011459
C02424=2156.343500,340.090900,-603.612600,91.054453,0.613065,0.011459
C02425=2142.360900,340.162400,-603.612600,91.020075,0.653172,0.011459
C02426=2153.966800,340.206100,-603.612600,90.957050,0.338045,0.005730
C02427=2118.636800,340.235500,-603.612600,90.802351,-0.292208,-0.005730
C02428=2076.694600,340.275700,-603.612600,91.300825,-1.019865,-0.022918
C02429=2112.962800,340.298400,-603.612600,90.670571,-0.744845,-0.011459
C02430=2144.168100,340.327100,-603.612600,91.346661,-0.223454,-0.005730
C02431=2061.348500,340.347700,-603.612600,91.134667,-0.355234,-0.005730
C02432=2073.181200,340.360500,-603.612600,90.922673,-1.002676,-0.017189
C02433=2167.096500,340.394700,-603.612600,90.613275,0.767763,0.005730
C02434=2135.276400,340.414600,-603.612600,90.733596,0.011459,0.000000
C02435=2108.758700,340.447700,-603.612600,91.358120,-0.756304,-0.017189
C02436=2167.455500,340.459200,-603.612600,90.309608,1.065701,0.005730
C02437=2072.723400,340.483500,-603.612600,90.103343,-0.561499,-0.000000
C02438=2170.625900,340.498000,-603.612600,90.424199,1.163104,0.011459
C02439=2120.756300,340.519700,-603.612600,90.997157,-0.234913,-0.005730
C02440=2089.944900,340.532500,-603.612600,91.111749,-0.595876,-0.011459
C02441=2055.163200,340.569300,-603.612600,91.123208,-0.607335,-0.011459
C02442=2155.478800,340.589300,-603.612600,90.258041,0.166158,0.000000
C02443=2081.867700,340.611600,-603.612600,91.340932,-0.309397,-0.005730
C02444=2166.000300,340.634500,-603.612600,90.401281,1.203211,0.005730
C02445=2093.938900,340.652800,-603.612600,90.762244,-0.509932,-0.005730
C02446=2069.645300,340.675800,-603.612600,91.661788,-1.254778,-0.034377
C02447=2178.852900,340.705500,-603.612600,90.235123,2.715820,0.011459
C02448=1874.120300,340.733500,-603.612600,91.117478,0.080214,0.000000
C02449=2167.772000,340.746400,-603.612600,89.484548,4.159674,-0.040107
C02450=2071.179200,340.784500,-603.612600,91.323743,-1.077161,-0.022918
C02451=2026.257800,340.804800,-603.612600,91.593033,0.177617,0.005730
C02452=2039.382400,340.810200,-603.612600,90.985698,-0.819330,-0.011459
C02453=1845.616200,340.815600,-603.612600,90.240853,-0.303668,-0.000000
C02454=2098.545900,340.841300,-603.612600,90.332526,-0.372423,-0.000000
C02455=1834.963300,340.847000,-603.612600,90.704949,0.005730,0.000000
C02456=2182.533600,340.865600,-603.612600,90.601816,2.394964,0.022918
C02457=1827.332900,340.906500,-603.612600,90.326796,-0.911003,-0.005730
C02458=2009.358000,340.930200,-603.612600,92.968132,0.796411,0.040107
C02459=1828.273600,340.940600,-603.612600,90.601816,-0.504203,-0.005730
C02460=2189.959500,340.945800,-603.612600,90.578898,-8.113082,-0.080214
C02461=1826.229800,340.967300,-603.612600,90.005940,-0.607335,-0.000000
C02462=2173.349000,340.985600,-603.612600,90.298149,1.690225,0.011459
C02463=1862.164100,340.998400,-603.612600,91.169044,0.744845,0.017189
C02464=1902.966300,341.006500,-603.612600,91.432605,0.527121,0.011459
C02465=1896.874400,341.026400,-603.612600,90.911213,0.630254,0.011459
C02466=1843.071100,341.041000,-603.612600,90.578898,-0.068755,-0.000000
C02467=1821.811600,341.061900,-603.612600,90.229394,-0.315127,-0.000000
C02468=2040.528500,341.073100,-603.612600,91.931078,-0.853707,-0.028648
C02469=2030.809300,341.086900,-603.612600,90.561709,-0.555769,-0.005730
C02470=1922.128600,341.098700,-603.612600,91.678977,0.234913,0.005730
C02471=1913.531000,341.101800,-603.612600,91.065912,0.429718,0.005730
C02472=1816.196200,341.117000,-603.612600,89.816864,-1.638659,0.005730
C02473=1892.901700,341.129100,-603.612600,91.283636,-0.131780,-0.005730
C02474=1855.602100,341.155800,-603.612600,90.567439,0.721927,0.005730
C02475=1813.245300,341.168300,-603.612600,89.398605,-1.128727,0.011459
C02476=2041.678700,341.179500,-603.612600,90.223664,-1.014135,-0.005730
C02477=2186.206500,341.193000,-603.612600,90.275230,-1.592823,-0.005730
C02478=1929.570000,341.202800,-603.612600,91.931078,0.584417,0.017189
C02479=1833.615100,341.217000,-603.612600,89.702272,0.716197,-0.005730
C02480=2020.591300,341.222700,-603.612600,91.650329,-0.481285,-0.011459
C02481=1884.225300,341.244700,-603.612600,90.722137,1.088620,0.011459
C02482=1898.398900,341.257200,-603.612600,91.163315,0.847978,0.017189
C02483=2014.799100,341.274100,-603.612600,91.524278,-0.194806,-0.005730
C02484=1908.938600,341.295000,-603.612600,90.928402,0.601606,0.011459
C02485=2004.014700,341.322100,-603.612600,91.054453,-0.956840,-0.017189
C02486=2007.317300,341.344700,-603.612600,91.936808,-1.082890,-0.034377
C02487=1886.600300,341.355500,-603.612600,91.083101,1.117268,0.022918
C02488=1870.568300,341.370400,-603.612600,90.974239,0.504203,0.005730
C02489=1934.460500,341.379800,-603.612600,91.243529,0.595876,0.011459
C02490=1959.958300,341.384600,-603.612600,91.323743,-0.257831,-0.005730
C02491=1799.058600,341.402900,-603.612600,90.017399,2.303290,0.000000
C02492=2016.771500,341.442300,-603.612600,91.123208,-0.246372,-0.005730
C02493=1973.170000,341.456900,-603.612600,92.045670,-0.641713,-0.022918
C02494=1987.390600,341.477100,-603.612600,90.905484,-0.395341,-0.005730
C02495=1944.689200,341.484900,-603.612600,91.684706,-0.143239,-0.005730
C02496=1886.880500,341.528800,-603.612600,91.157585,1.037054,0.022918
C02497=1896.840200,341.582500,-603.612600,91.031534,0.613065,0.011459
C02498=2036.002200,341.600800,-603.612600,90.298149,-1.002676,-0.005730
C02499=1926.992900,341.647400,-603.612600,91.535737,0.750575,0.022918
C02500=1904.287200,341.672700,-603.612600,91.163315,0.773493,0.017189
C02501=1922.547500,341.690600,-603.612600,91.318013,0.544310,0.011459
C02502=2010.209000,341.710600,-603.612600,91.042994,-0.813600,-0.017189
C02503=1993.488100,341.734200,-603.612600,90.957050,-0.171887,-0.000000
C02504=1988.105700,341.792300,-603.612600,90.802351,0.091673,0.000000
C02505=2019.868100,341.819000,-603.612600,90.601816,-0.423989,-0.005730
C02506=1974.252900,341.856500,-603.612600,91.879512,-0.618794,-0.022918
C02507=1935.427300,341.914000,-603.612600,91.203422,0.257831,0.005730
C02508=1994.529200,341.953500,-603.612600,91.340932,-0.148969,-0.005730
C02509=1978.104900,342.052500,-603.612600,92.355067,-0.842248,-0.034377
C02510=2001.864200,342.090100,-603.612600,90.704949,-1.249048,-0.017189
C02511=1961.792800,342.129500,-603.612600,90.905484,-0.280749,-0.005730
C02512=1968.211200,342.175300,-603.612600,91.174774,0.051566,0.000000
C02513=1995.375400,342.226800,-603.612600,90.315337,-0.269290,-0.000000
C02514=1959.702500,342.364300,-603.612600,91.375309,-0.275020,-0.005730
C02515=1799.585900,341.481900,-653.612600,89.862701,1.524068,-0.005730
C02516=1797.490800,341.408400,-653.612600,89.587681,4.703983,-0.034377
C02517=1798.072300,341.332900,-653.612600,89.547574,4.377398,-0.034377
C02518=1813.001800,341.180200,-653.612600,90.309608,-1.088620,-0.005730
C02519=1809.005700,341.137300,-653.612600,90.355444,-1.799087,-0.011459
C02520=1795.303000,341.117000,-653.612600,90.830999,12.931657,0.183346
C02521=1818.726600,341.080500,-653.612600,89.421523,-1.466772,0.017189
C02522=1939.900600,341.014300,-653.612600,91.678977,0.183346,0.005730
C02523=1794.649100,340.970000,-653.612600,91.191963,19.411810,0.395341
C02524=1920.963100,340.929100,-653.612600,90.429929,0.275020,0.000000
C02525=1993.976500,340.898400,-653.612600,91.615951,-0.693279,-0.017189
C02526=1907.219900,340.884200,-653.612600,91.455523,0.429718,0.011459
C02527=1822.301000,340.862600,-653.612600,90.435658,-1.191752,-0.011459
C02528=1952.703400,340.836900,-653.612600,91.885242,0.418259,0.011459
C02529=1900.084800,340.808500,-653.612600,90.292419,0.521392,0.000000
C02530=2005.588400,340.801800,-653.612600,91.169044,-0.297938,-0.005730
C02531=1920.569500,340.791600,-653.612600,91.805028,0.229183,0.005730
C02532=1993.982600,340.779800,-653.612600,94.108318,0.681820,0.051566
C02533=1964.959800,340.769200,-653.612600,93.867676,0.034377,0.000000
C02534=1960.912500,340.748700,-653.612600,90.429929,-0.183346,-0.000000
C02535=1944.714300,340.712200,-653.612600,90.578898,-0.234913,-0.000000
C02536=1861.279500,340.701400,-653.612600,91.736273,-0.538580,-0.017189
C02537=1877.044300,340.694500,-653.612600,90.596087,-0.704738,-0.005730
C02538=1851.847500,340.683500,-653.612600,90.275230,0.572958,0.000000
C02539=1848.928800,340.657800,-653.612600,90.286689,-0.343775,-0.000000
C02540=2186.041700,340.631500,-653.612600,90.240853,1.294885,0.005730
C02541=1837.769800,340.620000,-653.612600,90.212205,-0.893814,-0.005730
C02542=2179.220300,340.605900,-653.612600,89.988751,2.394964,-0.000000
C02543=2181.886700,340.594000,-653.612600,90.498684,2.864789,0.022918
C02544=1884.869400,340.587200,-653.612600,91.123208,0.366693,0.005730
C02545=1929.227100,340.579100,-653.612600,91.730543,0.028648,0.000000
C02546=1935.934100,340.554500,-653.612600,91.381039,0.423989,0.011459
C02547=1975.026200,340.541600,-653.612600,91.060182,0.091673,0.000000
C02548=1983.594200,340.531200,-653.612600,91.489901,-0.303668,-0.005730
C02549=1957.244600,340.515600,-653.612600,92.332149,-0.246372,-0.011459
C02550=2181.325200,340.501400,-653.612600,89.432982,2.647065,-0.028648
C02551=2029.531900,340.495000,-653.612600,91.358120,-0.567228,-0.011459
C02552=2008.733400,340.470900,-653.612600,90.177827,-0.888085,-0.000000
C02553=1931.404400,340.449100,-653.612600,90.974239,0.131780,0.000000
C02554=1879.484400,340.436600,-653.612600,90.452847,-0.091673,-0.000000
C02555=2187.220600,340.422500,-653.612600,92.458199,-2.085566,-0.091673
C02556=1907.734700,340.397400,-653.612600,90.470036,0.389611,0.005730
C02557=2042.416500,340.383900,-653.612600,91.461253,0.578687,0.017189
C02558=1896.512900,340.364600,-653.612600,90.504413,0.131780,0.000000
C02559=1863.838500,340.358500,-653.612600,90.464306,-0.223454,-0.000000
C02560=2027.516100,340.350600,-653.612600,90.922673,-0.807870,-0.011459
C02561=2190.389400,340.335200,-653.612600,92.280582,-12.650908,-0.498473
C02562=1857.257300,340.319000,-653.612600,90.544520,-0.635983,-0.005730
C02563=1871.454300,340.309200,-653.612600,90.303878,-0.343775,-0.000000
C02564=2172.656800,340.290000,-653.612600,89.948644,1.386558,-0.000000
C02565=2168.784800,340.287200,-653.612600,90.876836,1.088620,0.017189
C02566=1916.606900,340.274400,-653.612600,91.088830,0.108862,0.000000
C02567=1899.370000,340.264300,-653.612600,90.309608,-0.429718,-0.000000
C02568=2021.925500,340.239900,-653.612600,91.283636,-0.366693,-0.005730
C02569=1962.435200,340.223400,-653.612600,90.979968,0.126051,0.000000
C02570=1932.220400,340.197400,-653.612600,90.922673,0.005730,0.000000
C02571=2017.464600,340.184900,-653.612600,91.025805,0.051566,0.000000
C02572=2167.720400,340.167600,-653.612600,91.123208,0.641713,0.011459
C02573=1877.825700,340.144700,-653.612600,89.776757,-0.538580,0.000000
C02574=2038.197000,340.130600,-653.612600,90.670571,-0.257831,-0.005730
C02575=2080.355000,340.103100,-653.612600,90.447118,-0.114592,-0.000000
C02576=1931.894500,340.092300,-653.612600,90.945591,0.469825,0.005730
C02577=2072.300500,340.076400,-653.612600,91.386768,-0.217724,-0.005730
C02578=2165.460100,340.065300,-653.612600,90.384092,0.779223,0.005730
C02579=2065.765900,340.053800,-653.612600,90.607546,-0.057296,-0.000000
C02580=2148.257300,340.032200,-653.612600,90.796622,-0.280749,-0.005730
C02581=2048.677500,340.015200,-653.612600,90.160639,-0.360963,-0.000000
C02582=2152.310500,339.998700,-653.612600,88.355822,0.011459,-0.000000
C02583=2149.685900,339.989200,-653.612600,90.624734,0.572958,0.005730
C02584=1970.078100,339.973400,-653.612600,90.028858,0.435448,0.000000
C02585=2062.637900,339.953900,-653.612600,90.636194,0.223454,0.000000
C02586=2096.443900,339.933800,-653.612600,91.426875,0.028648,0.000000
C02587=2073.972100,339.918300,-653.612600,89.937185,-0.297938,0.000000
C02588=2130.009900,339.895700,-653.612600,90.510143,0.378152,0.005730
C02589=2162.184100,339.887900,-653.612600,90.040318,0.928192,0.000000
C02590=2087.105600,339.866600,-653.612600,90.636194,-0.303668,-0.005730
C02591=2156.929100,339.855100,-653.612600,89.639247,0.527121,-0.005730
C02592=2072.996200,339.844000,-653.612600,90.916943,0.108862,0.000000
C02593=2141.594800,339.830800,-653.612600,91.111749,1.598552,0.028648
C02594=2161.208200,339.821300,-653.612600,90.492954,1.008406,0.011459
C02595=2028.181600,339.808200,-653.612600,90.246582,-0.744845,-0.005730
C02596=2093.127500,339.781500,-653.612600,90.859647,-0.349504,-0.005730
C02597=2124.221900,339.766300,-653.612600,90.888295,0.040107,0.000000
C02598=2153.667000,339.747700,-653.612600,90.590357,0.618794,0.005730
C02599=2093.380700,339.739800,-653.612600,90.601816,-0.613065,-0.005730
C02600=2124.244200,339.722400,-653.612600,90.309608,0.217724,0.000000
C02601=2083.703800,339.682800,-653.612600,89.736650,-0.040107,0.000000
C02602=2127.061500,339.664600,-653.612600,89.885619,0.372423,-0.000000
C02603=2134.955000,339.649700,-653.612600,88.281337,0.951110,-0.028648
C02604=2101.613100,339.635500,-653.612600,90.263771,0.338045,0.000000
C02605=2118.165200,339.608800,-653.612600,90.544520,0.091673,0.000000
C02606=2116.317200,339.587900,-653.612600,90.957050,0.166158,0.000000
C02607=2128.394300,339.554800,-653.612600,90.934132,-0.097403,-0.000000
C02608=2114.039500,339.509200,-653.612600,90.653382,0.005730,0.000000
C02609=2073.190000,338.995300,-703.612600,90.515872,-0.108862,-0.000000
C02610=2063.755900,339.117900,-703.612600,90.767974,0.613065,0.005730
C02611=2093.591000,339.162900,-703.612600,90.343985,0.504203,0.005730
C02612=2077.013900,339.188600,-703.612600,89.215258,0.865166,-0.011459
C02613=2089.260300,339.222000,-703.612600,90.888295,0.847978,0.011459
C02614=1995.708200,339.241900,-703.612600,90.630464,-0.131780,-0.000000
C02615=2081.808100,339.252400,-703.612600,89.324120,0.962569,-0.011459
C02616=2023.063400,339.266900,-703.612600,90.533061,-0.063025,-0.000000
C02617=2029.208700,339.277400,-703.612600,89.776757,0.114592,-0.000000
C02618=1977.825400,339.286500,-703.612600,90.435658,-0.355234,-0.000000
C02619=2107.308000,339.308500,-703.612600,90.590357,-0.280749,-0.005730
C02620=2117.358700,339.319300,-703.612600,90.561709,0.126051,0.000000
C02621=2013.371800,339.330100,-703.612600,89.805405,-0.120321,0.000000
C02622=2059.863300,339.337500,-703.612600,90.492954,-0.063025,-0.000000
C02623=2048.126700,339.350700,-703.612600,90.916943,-0.057296,-0.000000
C02624=2083.336100,339.354800,-703.612600,90.951320,-0.171887,-0.005730
C02625=2037.648100,339.368600,-703.612600,90.332526,0.034377,0.000000
C02626=2099.786100,339.381500,-703.612600,89.839782,0.395341,-0.000000
C02627=2040.439600,339.396300,-703.612600,91.031534,-0.034377,-0.000000
C02628=1982.033500,339.410900,-703.612600,89.484548,-0.091673,0.000000
C02629=2066.113400,339.417300,-703.612600,90.573168,-0.567228,-0.005730
C02630=2130.776700,339.427400,-703.612600,89.874160,0.899544,-0.000000
C02631=2125.115200,339.438600,-703.612600,90.613275,-0.051566,-0.000000
C02632=2075.552700,339.453400,-703.612600,90.481495,-0.114592,-0.000000
C02633=2042.672400,339.464200,-703.612600,90.727867,0.418259,0.005730
C02634=2069.289400,339.474400,-703.612600,89.856971,0.166158,-0.000000
C02635=2058.758800,339.483200,-703.612600,90.332526,0.057296,0.000000
C02636=2057.580000,339.492600,-703.612600,90.011670,-1.071431,-0.000000
C02637=2134.466400,339.499700,-703.612600,89.690813,-0.171887,0.000000
C02638=2007.649000,339.513600,-703.612600,90.407010,-0.034377,-0.000000
C02639=2121.289900,339.520000,-703.612600,90.664842,0.022918,0.000000
C02640=2139.914800,339.533800,-703.612600,90.028858,0.613065,0.000000
C02641=2048.001400,339.547000,-703.612600,90.533061,-0.509932,-0.005730
C02642=2190.966300,339.567600,-703.612600,90.114802,-14.587505,-0.028648
C02643=2134.176000,339.577400,-703.612600,90.286689,0.028648,0.000000
C02644=2149.575100,339.602400,-703.612600,89.851241,0.607335,-0.000000
C02645=2146.144700,339.608500,-703.612600,90.458577,0.401070,0.005730
C02646=2154.030200,339.619600,-703.612600,90.624734,-0.515662,-0.005730
C02647=2156.547400,339.633500,-703.612600,90.263771,0.756304,0.005730
C02648=1911.745800,339.643600,-703.612600,89.587681,-0.710468,0.005730
C02649=1997.455300,339.656100,-703.612600,91.146126,-0.509932,-0.011459
C02650=1962.991900,339.666400,-703.612600,90.676301,-0.401070,-0.005730
C02651=2020.153500,339.671700,-703.612600,92.481118,0.028648,0.000000
C02652=2151.746500,339.683800,-703.612600,90.280960,0.389611,0.000000
C02653=1978.709600,339.695000,-703.612600,91.530008,-0.481285,-0.011459
C02654=2191.127700,339.708200,-703.612600,91.123208,-14.054655,-0.275020
C02655=2163.110900,339.716900,-703.612600,90.504413,0.389611,0.005730
C02656=1903.782200,339.744000,-703.612600,90.137720,-0.647442,-0.000000
C02657=1940.902300,339.759900,-703.612600,90.561709,-0.022918,-0.000000
C02658=2183.988700,339.776800,-703.612600,90.492954,-0.338045,-0.005730
C02659=1960.082100,339.794700,-703.612600,90.825270,-0.171887,-0.000000
C02660=1883.595100,339.814900,-703.612600,89.839782,-0.813600,0.000000
C02661=1912.900100,339.833200,-703.612600,90.756515,-0.074485,-0.000000
C02662=2178.615900,339.846900,-703.612600,90.074695,1.340721,0.000000
C02663=2024.628200,339.859500,-703.612600,90.945591,-0.257831,-0.005730
C02664=2178.476200,339.872400,-703.612600,92.320690,-0.309397,-0.011459
C02665=2183.640900,339.884900,-703.612600,91.530008,2.687172,0.074485
C02666=2174.707300,339.907200,-703.612600,91.352391,1.300614,0.028648
C02667=1897.922100,339.912900,-703.612600,89.335579,0.504203,-0.005730
C02668=1933.132200,339.928100,-703.612600,90.974239,-0.022918,-0.000000
C02669=1878.689400,339.963200,-703.612600,90.212205,-1.157375,-0.005730
C02670=1895.861200,339.983200,-703.612600,90.664842,-0.103132,-0.000000
C02671=1902.499900,340.024700,-703.612600,91.759191,0.372423,0.011459
C02672=1936.508900,340.046300,-703.612600,90.733596,0.807870,0.011459
C02673=1947.976400,340.058500,-703.612600,90.888295,-0.137510,-0.000000
C02674=1883.597900,340.066300,-703.612600,90.292419,-0.888085,-0.005730
C02675=2183.839600,340.085500,-703.612600,90.842458,2.137133,0.028648
C02676=1917.888200,340.119000,-703.612600,90.292419,0.166158,0.000000
C02677=1873.671400,340.134900,-703.612600,90.068965,-0.481285,-0.000000
C02678=2183.708500,340.173000,-703.612600,90.074695,0.853707,0.000000
C02679=1859.955700,340.209500,-703.612600,90.441388,-1.518338,-0.011459
C02680=1876.642400,340.250100,-703.612600,90.733596,-0.492744,-0.005730
C02681=2185.258800,340.280100,-703.612600,91.094560,0.068755,0.000000
C02682=1857.611600,340.327300,-703.612600,89.627788,-0.527121,0.005730
C02683=1852.308600,340.478500,-703.612600,89.742379,-1.283425,0.005730
C02684=1844.337800,340.522700,-703.612600,90.068965,-0.813600,-0.000000
C02685=1839.074000,340.629800,-703.612600,90.160639,-1.163104,-0.005730
C02686=1828.744200,340.737200,-703.612600,89.725191,-0.315127,0.000000
C02687=1825.416300,340.774700,-703.612600,90.292419,-0.750575,-0.005730
C02688=1794.825500,340.931200,-703.612600,89.622058,19.308678,-0.126051
C02689=1816.931300,341.031700,-703.612600,89.656436,-1.214671,0.005730
C02690=1818.991900,341.110600,-703.612600,89.771027,-1.976704,0.005730
C02691=1795.182400,341.178100,-703.612600,85.955128,15.985522,-1.117268
C02692=1805.178300,341.310900,-703.612600,89.559033,-1.535527,0.011459
C02693=1809.277200,341.405200,-703.612600,89.243906,-1.449583,0.017189
C02694=1798.100500,341.483700,-703.612600,88.848565,4.348750,-0.085944
C02695=1799.488700,341.555200,-703.612600,90.384092,0.131780,0.000000
C02696=1799.967800,341.624600,-753.612600,90.395551,1.168834,0.005730
C02697=1803.673700,341.530200,-753.612600,91.111749,-1.604282,-0.028648
C02698=1804.957300,341.437600,-753.612600,88.670948,-0.979758,0.022918
C02699=1807.130900,341.404100,-753.612600,89.667895,-1.077161,0.005730
C02700=1813.473700,341.329500,-753.612600,89.730920,-1.174563,0.005730
C02701=1810.931100,341.258900,-753.612600,90.005940,-1.701685,-0.000000
C02702=1820.076200,341.165000,-753.612600,90.263771,-0.464096,-0.000000
C02703=1829.211600,341.091300,-753.612600,90.326796,-0.979758,-0.005730
C02704=1827.450400,340.976400,-753.612600,89.748109,-1.271966,0.005730
C02705=1827.531900,340.915600,-753.612600,90.515872,-0.784952,-0.005730
C02706=1841.303000,340.791000,-753.612600,89.547574,-1.186023,0.011459
C02707=1844.090600,340.649700,-753.612600,89.679354,-1.306344,0.005730
C02708=1848.833300,340.492000,-753.612600,89.885619,-1.409476,0.000000
C02709=1855.718800,340.392000,-753.612600,89.427253,-1.071431,0.011459
C02710=1859.766500,340.307500,-753.612600,89.988751,-1.501149,0.000000
C02711=1862.410900,340.204500,-753.612600,89.960103,-1.816276,0.000000
C02712=1863.830900,340.143000,-753.612600,89.478819,-1.357910,0.011459
C02713=1881.470100,340.082500,-753.612600,89.971563,-0.429718,0.000000
C02714=1887.120200,340.005600,-753.612600,89.530385,-0.401070,0.005730
C02715=1889.231100,339.927400,-753.612600,89.914267,-0.303668,0.000000
C02716=1888.561600,339.891600,-753.612600,90.120532,-1.334992,-0.000000
C02717=1902.175100,339.843600,-753.612600,90.057506,-0.320856,-0.000000
C02718=1899.627200,339.779400,-753.612600,90.292419,-0.865166,-0.005730
C02719=1897.177300,339.749000,-753.612600,89.685084,-0.498473,0.000000
C02720=2160.074300,339.715900,-753.612600,90.366903,0.057296,0.000000
C02721=1899.047900,339.686200,-753.612600,89.581951,-0.406800,0.005730
C02722=2191.473800,339.658800,-753.612600,89.856971,-17.927849,0.045837
C02723=1908.888700,339.625700,-753.612600,90.258041,-0.658901,-0.005730
C02724=2178.824500,339.612400,-753.612600,89.742379,1.226130,-0.005730
C02725=1918.495400,339.594000,-753.612600,89.696543,-0.515662,0.000000
C02726=2163.106000,339.570700,-753.612600,90.533061,0.160428,0.000000
C02727=2163.901400,339.560900,-753.612600,90.034588,-0.527121,-0.000000
C02728=1918.974900,339.531800,-753.612600,90.292419,-0.269290,-0.000000
C02729=2179.564000,339.514900,-753.612600,90.412740,1.008406,0.005730
C02730=2153.582000,339.502100,-753.612600,90.785163,0.160428,0.000000
C02731=1927.798400,339.497000,-753.612600,89.708002,-0.721927,0.005730
C02732=1963.372400,339.484200,-753.612600,90.429929,-0.813600,-0.005730
C02733=2153.419600,339.472000,-753.612600,90.343985,0.343775,0.000000
C02734=1924.024300,339.462200,-753.612600,90.109072,-0.670361,-0.000000
C02735=2168.128500,339.440600,-753.612600,89.811134,-0.263561,0.000000
C02736=2127.752000,339.424400,-753.612600,89.644977,0.406800,-0.000000
C02737=2157.929600,339.408800,-753.612600,90.131991,0.458366,0.000000
C02738=2182.084600,339.396000,-753.612600,89.415794,1.140186,-0.011459
C02739=1943.022500,339.384800,-753.612600,90.590357,-0.676090,-0.005730
C02740=1943.388800,339.372700,-753.612600,89.891348,-0.825059,0.000000
C02741=2146.933500,339.357800,-753.612600,90.212205,0.223454,0.000000
C02742=1944.277600,339.339600,-753.612600,89.730920,-0.194806,0.000000
C02743=2145.381100,339.321700,-753.612600,90.561709,0.263561,0.000000
C02744=1955.529700,339.311500,-753.612600,90.429929,-0.097403,-0.000000
C02745=2126.821700,339.291900,-753.612600,90.607546,0.183346,0.000000
C02746=1946.430600,339.286200,-753.612600,89.702272,-0.234913,0.000000
C02747=1963.293300,339.277100,-753.612600,88.968886,-0.423989,0.005730
C02748=1985.309500,339.259500,-753.612600,91.226340,-0.452637,-0.011459
C02749=1961.859400,339.246000,-753.612600,91.191963,-0.567228,-0.011459
C02750=2133.264900,339.234800,-753.612600,89.788216,0.882355,-0.005730
C02751=2001.200700,339.224400,-753.612600,90.034588,0.166158,0.000000
C02752=1953.498000,339.214900,-753.612600,90.005940,0.229183,0.000000
C02753=2110.513300,339.208100,-753.612600,89.679354,0.492744,-0.000000
C02754=2010.070900,339.200700,-753.612600,90.538791,-0.607335,-0.005730
C02755=2133.135300,339.191600,-753.612600,90.894025,0.538580,0.005730
C02756=2014.725900,339.180100,-753.612600,90.361174,0.040107,0.000000
C02757=2125.637000,339.165600,-753.612600,90.298149,-0.114592,-0.000000
C02758=2104.683100,339.146700,-753.612600,90.343985,0.303668,0.000000
C02759=2129.776300,339.141300,-753.612600,90.154909,0.807870,0.000000
C02760=2071.817400,339.136900,-753.612600,91.134667,0.280749,0.005730
C02761=2057.477500,339.112500,-753.612600,89.610599,1.375099,-0.011459
C02762=2061.228900,339.100400,-753.612600,90.269501,-0.068755,-0.000000
C02763=1975.866400,339.086500,-753.612600,90.905484,-0.166158,-0.000000
C02764=2041.824700,339.079400,-753.612600,90.796622,-0.040107,-0.000000
C02765=2058.845200,339.075000,-753.612600,90.407010,0.813600,0.005730
C02766=2015.305100,339.069600,-753.612600,89.736650,-1.088620,0.005730
C02767=1968.919900,339.056800,-753.612600,91.254988,-0.504203,-0.011459
C02768=2054.725400,339.041300,-753.612600,90.355444,0.297938,0.000000
